   DATA[1768,11] := 19.63634;
   DATA[1768,12] := 2.208884;
   DATA[1768,13] := 823.5469;
   DATA[1768,14] := 1.0;
   DATA[1768,15] := 2.0;
   DATA[1768,16] := 1.0;
   DATA[1768,17] := 1.0;
   DATA[1768,18] := 1.0;
   DATA[1768,19] := 2.0;
   DATA[1768,20] := 148.808;
   DATA[1768,21] := 154.4219;
   DATA[1768,22] := 1.717105;
   DATA[1768,23] := 810.9075;
   DATA[1768,24] := 2.0;
   DATA[1768,25] := 2.0;
   DATA[1768,26] := 7.876058;
   DATA[1768,27] := 143.7067;
   DATA[1768,28] := 262.4007;
   DATA[1768,29] := 12.11228;
   DATA[1768,30] := 1.725455;
   DATA[1768,31] := 1.290124;
   DATA[1768,32] := 0.7353967;
   DATA[1768,33] := 0.3080421;
   DATA[1768,34] := 2.0;
   DATA[1768,35] := 250.1923;
   DATA[1768,36] := 1.681991;
   DATA[1768,37] := 188.974;
   DATA[1768,38] := 0.000128152;
   DATA[1768,39] := 1.0;
   DATA[1768,40] := 1.0;
   DATA[1769,0] := 2.554847;
   DATA[1769,1] := 822.777;
   DATA[1769,2] := 2.0;
   DATA[1769,3] := 1.0;
   DATA[1769,4] := 262.625;
   DATA[1769,5] := 8.46533;
   DATA[1769,6] := 319.7898;
   DATA[1769,8] := 1.0;
   DATA[1769,9] := 1.0;
   DATA[1769,10] := 1.0;
   DATA[1769,11] := 19.70037;
   DATA[1769,12] := 2.208884;
   DATA[1769,13] := 823.3466;
   DATA[1769,14] := 1.0;
   DATA[1769,15] := 2.0;
   DATA[1769,16] := 1.0;
   DATA[1769,17] := 1.0;
   DATA[1769,18] := 1.0;
   DATA[1769,19] := 2.0;
   DATA[1769,20] := 148.808;
   DATA[1769,21] := 154.4219;
   DATA[1769,22] := 1.717105;
   DATA[1769,23] := 810.6383;
   DATA[1769,24] := 2.0;
   DATA[1769,25] := 2.0;
   DATA[1769,26] := 7.876058;
   DATA[1769,27] := 143.7067;
   DATA[1769,28] := 262.4007;
   DATA[1769,29] := 12.11228;
   DATA[1769,30] := 1.725455;
   DATA[1769,31] := 1.291533;
   DATA[1769,32] := 0.7353967;
   DATA[1769,33] := 0.3083624;
   DATA[1769,34] := 2.0;
   DATA[1769,35] := 250.1923;
   DATA[1769,36] := 1.681991;
   DATA[1769,37] := 188.974;
   DATA[1769,38] := 0.000128152;
   DATA[1769,39] := 1.0;
   DATA[1769,40] := 1.0;
   DATA[1770,0] := 2.542036;
   DATA[1770,1] := 823.0518;
   DATA[1770,2] := 2.0;
   DATA[1770,3] := 1.0;
   DATA[1770,4] := 262.625;
   DATA[1770,5] := 8.46533;
   DATA[1770,6] := 319.7898;
   DATA[1770,8] := 1.0;
   DATA[1770,9] := 1.0;
   DATA[1770,10] := 1.0;
   DATA[1770,11] := 19.73558;
   DATA[1770,12] := 2.208884;
   DATA[1770,13] := 823.0262;
   DATA[1770,14] := 1.0;
   DATA[1770,15] := 2.0;
   DATA[1770,16] := 1.0;
   DATA[1770,17] := 1.0;
   DATA[1770,18] := 1.0;
   DATA[1770,19] := 2.0;
   DATA[1770,20] := 148.808;
   DATA[1770,21] := 154.3707;
   DATA[1770,22] := 1.717105;
   DATA[1770,23] := 811.0228;
   DATA[1770,24] := 2.0;
   DATA[1770,25] := 2.0;
   DATA[1770,26] := 7.876058;
   DATA[1770,27] := 143.5529;
   DATA[1770,28] := 262.4007;
   DATA[1770,29] := 12.11228;
   DATA[1770,30] := 1.725455;
   DATA[1770,31] := 1.291533;
   DATA[1770,32] := 0.7353967;
   DATA[1770,33] := 0.3084265;
   DATA[1770,34] := 2.0;
   DATA[1770,35] := 250.1923;
   DATA[1770,36] := 1.681991;
   DATA[1770,37] := 188.974;
   DATA[1770,38] := 0.000128152;
   DATA[1770,39] := 1.0;
   DATA[1770,40] := 1.0;
   DATA[1771,0] := 2.526022;
   DATA[1771,1] := 823.7976;
   DATA[1771,2] := 2.0;
   DATA[1771,3] := 1.0;
   DATA[1771,4] := 262.625;
   DATA[1771,5] := 8.46533;
   DATA[1771,6] := 319.7898;
   DATA[1771,8] := 1.0;
   DATA[1771,9] := 1.0;
   DATA[1771,10] := 1.0;
   DATA[1771,11] := 19.73558;
   DATA[1771,12] := 2.208884;
   DATA[1771,13] := 822.6657;
   DATA[1771,14] := 1.0;
   DATA[1771,15] := 2.0;
   DATA[1771,16] := 1.0;
   DATA[1771,17] := 1.0;
   DATA[1771,18] := 1.0;
   DATA[1771,19] := 2.0;
   DATA[1771,20] := 148.808;
   DATA[1771,21] := 154.3194;
   DATA[1771,22] := 1.716208;
   DATA[1771,23] := 810.9459;
   DATA[1771,24] := 2.0;
   DATA[1771,25] := 2.0;
   DATA[1771,26] := 7.876058;
   DATA[1771,27] := 143.5529;
   DATA[1771,28] := 262.4007;
   DATA[1771,29] := 12.11228;
   DATA[1771,30] := 1.725455;
   DATA[1771,31] := 1.291533;
   DATA[1771,32] := 0.7353967;
   DATA[1771,33] := 0.3084265;
   DATA[1771,34] := 2.0;
   DATA[1771,35] := 250.1923;
   DATA[1771,36] := 1.681991;
   DATA[1771,37] := 188.974;
   DATA[1771,38] := 0.000128152;
   DATA[1771,39] := 1.0;
   DATA[1771,40] := 1.0;
   DATA[1772,0] := 2.503923;
   DATA[1772,1] := 824.5042;
   DATA[1772,2] := 2.0;
   DATA[1772,3] := 1.0;
   DATA[1772,4] := 262.625;
   DATA[1772,5] := 8.46533;
   DATA[1772,6] := 319.7898;
   DATA[1772,8] := 1.0;
   DATA[1772,9] := 1.0;
   DATA[1772,10] := 1.0;
   DATA[1772,11] := 19.73558;
   DATA[1772,12] := 2.208884;
   DATA[1772,13] := 822.3853;
   DATA[1772,14] := 1.0;
   DATA[1772,15] := 2.0;
   DATA[1772,16] := 1.0;
   DATA[1772,17] := 1.0;
   DATA[1772,18] := 1.0;
   DATA[1772,19] := 2.0;
   DATA[1772,20] := 148.808;
   DATA[1772,21] := 154.2425;
   DATA[1772,22] := 1.715183;
   DATA[1772,23] := 811.4843;
   DATA[1772,24] := 2.0;
   DATA[1772,25] := 2.0;
   DATA[1772,26] := 7.876058;
   DATA[1772,27] := 143.5529;
   DATA[1772,28] := 262.4007;
   DATA[1772,29] := 12.11228;
   DATA[1772,30] := 1.723789;
   DATA[1772,31] := 1.282567;
   DATA[1772,32] := 0.7353967;
   DATA[1772,33] := 0.3084265;
   DATA[1772,34] := 2.0;
   DATA[1772,35] := 250.1923;
   DATA[1772,36] := 1.681991;
   DATA[1772,37] := 188.974;
   DATA[1772,38] := 0.000128152;
   DATA[1772,39] := 1.0;
   DATA[1772,40] := 1.0;
   DATA[1773,0] := 2.491432;
   DATA[1773,1] := 824.5042;
   DATA[1773,2] := 2.0;
   DATA[1773,3] := 1.0;
   DATA[1773,4] := 262.625;
   DATA[1773,5] := 8.46533;
   DATA[1773,6] := 319.7898;
   DATA[1773,8] := 1.0;
   DATA[1773,9] := 1.0;
   DATA[1773,10] := 1.0;
   DATA[1773,11] := 19.73558;
   DATA[1773,12] := 2.208884;
   DATA[1773,13] := 821.6643;
   DATA[1773,14] := 1.0;
   DATA[1773,15] := 2.0;
   DATA[1773,16] := 1.0;
   DATA[1773,17] := 1.0;
   DATA[1773,18] := 1.0;
   DATA[1773,19] := 2.0;
   DATA[1773,20] := 148.808;
   DATA[1773,21] := 154.2425;
   DATA[1773,22] := 1.715183;
   DATA[1773,23] := 811.3304;
   DATA[1773,24] := 2.0;
   DATA[1773,25] := 2.0;
   DATA[1773,26] := 7.876058;
   DATA[1773,27] := 143.5529;
   DATA[1773,28] := 262.4007;
   DATA[1773,29] := 12.11228;
   DATA[1773,30] := 1.723789;
   DATA[1773,31] := 1.266171;
   DATA[1773,32] := 0.7353967;
   DATA[1773,33] := 0.3084265;
   DATA[1773,34] := 2.0;
   DATA[1773,35] := 250.1923;
   DATA[1773,36] := 1.681991;
   DATA[1773,37] := 188.974;
   DATA[1773,38] := 0.000128152;
   DATA[1773,39] := 1.0;
   DATA[1773,40] := 1.0;
   DATA[1774,0] := 2.475098;
   DATA[1774,1] := 824.936;
   DATA[1774,2] := 2.0;
   DATA[1774,3] := 1.0;
   DATA[1774,4] := 262.625;
   DATA[1774,5] := 8.46533;
   DATA[1774,6] := 319.7898;
   DATA[1774,8] := 1.0;
   DATA[1774,9] := 1.0;
   DATA[1774,10] := 1.0;
   DATA[1774,11] := 19.73558;
   DATA[1774,12] := 2.208884;
   DATA[1774,13] := 821.8245;
   DATA[1774,14] := 1.0;
   DATA[1774,15] := 2.0;
   DATA[1774,16] := 1.0;
   DATA[1774,17] := 1.0;
   DATA[1774,18] := 1.0;
   DATA[1774,19] := 2.0;
   DATA[1774,20] := 148.808;
   DATA[1774,21] := 154.2425;
   DATA[1774,22] := 1.715183;
   DATA[1774,23] := 811.4073;
   DATA[1774,24] := 2.0;
   DATA[1774,25] := 2.0;
   DATA[1774,26] := 7.876058;
   DATA[1774,27] := 143.5529;
   DATA[1774,28] := 262.4007;
   DATA[1774,29] := 12.11228;
   DATA[1774,30] := 1.723789;
   DATA[1774,31] := 1.266299;
   DATA[1774,32] := 0.7353967;
   DATA[1774,33] := 0.3084265;
   DATA[1774,34] := 2.0;
   DATA[1774,35] := 250.032;
   DATA[1774,36] := 1.681991;
   DATA[1774,37] := 188.974;
   DATA[1774,38] := 0.000128152;
   DATA[1774,39] := 1.0;
   DATA[1774,40] := 1.0;
   DATA[1775,0] := 2.455241;
   DATA[1775,1] := 825.2892;
   DATA[1775,2] := 2.0;
   DATA[1775,3] := 1.0;
   DATA[1775,4] := 262.625;
   DATA[1775,5] := 8.46533;
   DATA[1775,6] := 319.7898;
   DATA[1775,8] := 1.0;
   DATA[1775,9] := 1.0;
   DATA[1775,10] := 1.0;
   DATA[1775,11] := 19.74198;
   DATA[1775,12] := 2.208884;
   DATA[1775,13] := 821.0235;
   DATA[1775,14] := 1.0;
   DATA[1775,15] := 2.0;
   DATA[1775,16] := 1.0;
   DATA[1775,17] := 1.0;
   DATA[1775,18] := 1.0;
   DATA[1775,19] := 2.0;
   DATA[1775,20] := 148.808;
   DATA[1775,21] := 154.5245;
   DATA[1775,22] := 1.715183;
   DATA[1775,23] := 811.4843;
   DATA[1775,24] := 2.0;
   DATA[1775,25] := 2.0;
   DATA[1775,26] := 7.876058;
   DATA[1775,27] := 143.5529;
   DATA[1775,28] := 262.4007;
   DATA[1775,29] := 12.11228;
   DATA[1775,30] := 1.723789;
   DATA[1775,31] := 1.260664;
   DATA[1775,32] := 0.7353967;
   DATA[1775,33] := 0.3084265;
   DATA[1775,34] := 2.0;
   DATA[1775,35] := 250.032;
   DATA[1775,36] := 1.762086;
   DATA[1775,37] := 188.9259;
   DATA[1775,38] := 0.000128152;
   DATA[1775,39] := 1.0;
   DATA[1775,40] := 1.0;
   DATA[1776,0] := 2.441149;
   DATA[1776,1] := 825.3677;
   DATA[1776,2] := 2.0;
   DATA[1776,3] := 1.0;
   DATA[1776,4] := 262.625;
   DATA[1776,5] := 8.46533;
   DATA[1776,6] := 319.7898;
   DATA[1776,8] := 1.0;
   DATA[1776,9] := 1.0;
   DATA[1776,10] := 1.0;
   DATA[1776,11] := 19.82201;
   DATA[1776,12] := 2.209013;
   DATA[1776,13] := 820.5428;
   DATA[1776,14] := 1.0;
   DATA[1776,15] := 2.0;
   DATA[1776,16] := 1.0;
   DATA[1776,17] := 1.0;
   DATA[1776,18] := 1.0;
   DATA[1776,19] := 2.0;
   DATA[1776,20] := 148.808;
   DATA[1776,21] := 154.5245;
   DATA[1776,22] := 1.718002;
   DATA[1776,23] := 811.1766;
   DATA[1776,24] := 2.0;
   DATA[1776,25] := 2.0;
   DATA[1776,26] := 7.876058;
   DATA[1776,27] := 143.5529;
   DATA[1776,28] := 262.5288;
   DATA[1776,29] := 12.11228;
   DATA[1776,30] := 1.723789;
   DATA[1776,31] := 1.265787;
   DATA[1776,32] := 0.7353967;
   DATA[1776,33] := 0.3084265;
   DATA[1776,34] := 2.0;
   DATA[1776,35] := 250.032;
   DATA[1776,36] := 1.810143;
   DATA[1776,37] := 188.9259;
   DATA[1776,38] := 0.000128152;
   DATA[1776,39] := 1.0;
   DATA[1776,40] := 1.0;
   DATA[1777,0] := 2.428658;
   DATA[1777,1] := 825.9173;
   DATA[1777,2] := 2.0;
   DATA[1777,3] := 1.0;
   DATA[1777,4] := 262.625;
   DATA[1777,5] := 8.46533;
   DATA[1777,6] := 319.7898;
   DATA[1777,8] := 1.0;
   DATA[1777,9] := 1.0;
   DATA[1777,10] := 1.0;
   DATA[1777,11] := 19.84762;
   DATA[1777,12] := 2.209013;
   DATA[1777,13] := 820.0622;
   DATA[1777,14] := 1.0;
   DATA[1777,15] := 2.0;
   DATA[1777,16] := 1.0;
   DATA[1777,17] := 1.0;
   DATA[1777,18] := 1.0;
   DATA[1777,19] := 2.0;
   DATA[1777,20] := 148.808;
   DATA[1777,21] := 154.5245;
   DATA[1777,22] := 1.718002;
   DATA[1777,23] := 811.5227;
   DATA[1777,24] := 2.0;
   DATA[1777,25] := 2.0;
   DATA[1777,26] := 7.876058;
   DATA[1777,27] := 143.5529;
   DATA[1777,28] := 262.5288;
   DATA[1777,29] := 12.11228;
   DATA[1777,30] := 1.723789;
   DATA[1777,31] := 1.267196;
   DATA[1777,32] := 0.7353967;
   DATA[1777,33] := 0.3084265;
   DATA[1777,34] := 2.0;
   DATA[1777,35] := 250.032;
   DATA[1777,36] := 1.810143;
   DATA[1777,37] := 188.9259;
   DATA[1777,38] := 0.000128152;
   DATA[1777,39] := 1.0;
   DATA[1777,40] := 1.0;
   DATA[1778,0] := 2.425135;
   DATA[1778,1] := 826.3491;
   DATA[1778,2] := 2.0;
   DATA[1778,3] := 1.0;
   DATA[1778,4] := 262.625;
   DATA[1778,5] := 8.46533;
   DATA[1778,6] := 319.7898;
   DATA[1778,8] := 1.0;
   DATA[1778,9] := 1.0;
   DATA[1778,10] := 1.0;
   DATA[1778,11] := 19.84762;
   DATA[1778,12] := 2.209525;
   DATA[1778,13] := 819.6216;
   DATA[1778,14] := 1.0;
   DATA[1778,15] := 2.0;
   DATA[1778,16] := 1.0;
   DATA[1778,17] := 1.0;
   DATA[1778,18] := 1.0;
   DATA[1778,19] := 2.0;
   DATA[1778,20] := 148.808;
   DATA[1778,21] := 154.5245;
   DATA[1778,22] := 1.718002;
   DATA[1778,23] := 811.0997;
   DATA[1778,24] := 2.0;
   DATA[1778,25] := 2.0;
   DATA[1778,26] := 7.876058;
   DATA[1778,27] := 143.5529;
   DATA[1778,28] := 262.5288;
   DATA[1778,29] := 12.11228;
   DATA[1778,30] := 1.723789;
   DATA[1778,31] := 1.262969;
   DATA[1778,32] := 0.7353967;
   DATA[1778,33] := 0.3084265;
   DATA[1778,34] := 2.0;
   DATA[1778,35] := 250.032;
   DATA[1778,36] := 1.810143;
   DATA[1778,37] := 188.9259;
   DATA[1778,38] := 0.000128152;
   DATA[1778,39] := 1.0;
   DATA[1778,40] := 1.0;
   DATA[1779,0] := 2.425135;
   DATA[1779,1] := 826.6631;
   DATA[1779,2] := 2.0;
   DATA[1779,3] := 1.0;
   DATA[1779,4] := 262.625;
   DATA[1779,5] := 8.46533;
   DATA[1779,6] := 319.7898;
   DATA[1779,8] := 1.0;
   DATA[1779,9] := 1.0;
   DATA[1779,10] := 1.0;
   DATA[1779,11] := 19.7836;
   DATA[1779,12] := 2.209525;
   DATA[1779,13] := 819.0208;
   DATA[1779,14] := 1.0;
   DATA[1779,15] := 2.0;
   DATA[1779,16] := 1.0;
   DATA[1779,17] := 1.0;
   DATA[1779,18] := 1.0;
   DATA[1779,19] := 2.0;
   DATA[1779,20] := 148.808;
   DATA[1779,21] := 154.5245;
   DATA[1779,22] := 1.718002;
   DATA[1779,23] := 810.7921;
   DATA[1779,24] := 2.0;
   DATA[1779,25] := 2.0;
   DATA[1779,26] := 7.876058;
   DATA[1779,27] := 143.5529;
   DATA[1779,28] := 262.5288;
   DATA[1779,29] := 12.11228;
   DATA[1779,30] := 1.723789;
   DATA[1779,31] := 1.267452;
   DATA[1779,32] := 0.7353967;
   DATA[1779,33] := 0.3084265;
   DATA[1779,34] := 2.0;
   DATA[1779,35] := 250.032;
   DATA[1779,36] := 1.665972;
   DATA[1779,37] := 188.9259;
   DATA[1779,38] := 0.000128152;
   DATA[1779,39] := 1.0;
   DATA[1779,40] := 1.0;
   DATA[1780,0] := 2.43026;
   DATA[1780,1] := 827.8799;
   DATA[1780,2] := 2.0;
   DATA[1780,3] := 1.0;
   DATA[1780,4] := 262.625;
   DATA[1780,5] := 8.46533;
   DATA[1780,6] := 319.7898;
   DATA[1780,8] := 1.0;
   DATA[1780,9] := 1.0;
   DATA[1780,10] := 1.0;
   DATA[1780,11] := 19.73558;
   DATA[1780,12] := 2.209525;
   DATA[1780,13] := 819.1409;
   DATA[1780,14] := 1.0;
   DATA[1780,15] := 2.0;
   DATA[1780,16] := 1.0;
   DATA[1780,17] := 1.0;
   DATA[1780,18] := 1.0;
   DATA[1780,19] := 2.0;
   DATA[1780,20] := 148.808;
   DATA[1780,21] := 154.5245;
   DATA[1780,22] := 1.715952;
   DATA[1780,23] := 811.0228;
   DATA[1780,24] := 2.0;
   DATA[1780,25] := 2.0;
   DATA[1780,26] := 7.876058;
   DATA[1780,27] := 143.5529;
   DATA[1780,28] := 262.5288;
   DATA[1780,29] := 12.11228;
   DATA[1780,30] := 1.723789;
   DATA[1780,31] := 1.28103;
   DATA[1780,32] := 0.7353967;
   DATA[1780,33] := 0.3084265;
   DATA[1780,34] := 2.0;
   DATA[1780,35] := 250.032;
   DATA[1780,36] := 1.665972;
   DATA[1780,37] := 188.8458;
   DATA[1780,38] := 0.000128152;
   DATA[1780,39] := 1.0;
   DATA[1780,40] := 1.0;
   DATA[1781,0] := 2.483105;
   DATA[1781,1] := 828.7042;
   DATA[1781,2] := 2.0;
   DATA[1781,3] := 1.0;
   DATA[1781,4] := 262.625;
   DATA[1781,5] := 8.46533;
   DATA[1781,6] := 319.7898;
   DATA[1781,8] := 1.0;
   DATA[1781,9] := 1.0;
   DATA[1781,10] := 1.0;
   DATA[1781,11] := 19.73558;
   DATA[1781,12] := 2.209525;
   DATA[1781,13] := 818.42;
   DATA[1781,14] := 1.0;
   DATA[1781,15] := 2.0;
   DATA[1781,16] := 1.0;
   DATA[1781,17] := 1.0;
   DATA[1781,18] := 1.0;
   DATA[1781,19] := 2.0;
   DATA[1781,20] := 148.808;
   DATA[1781,21] := 154.5245;
   DATA[1781,22] := 1.715952;
   DATA[1781,23] := 810.8306;
   DATA[1781,24] := 2.0;
   DATA[1781,25] := 2.0;
   DATA[1781,26] := 7.876058;
   DATA[1781,27] := 143.5529;
   DATA[1781,28] := 262.5288;
   DATA[1781,29] := 12.11228;
   DATA[1781,30] := 1.721738;
   DATA[1781,31] := 1.28167;
   DATA[1781,32] := 0.7353967;
   DATA[1781,33] := 0.3084265;
   DATA[1781,34] := 2.0;
   DATA[1781,35] := 250.032;
   DATA[1781,36] := 1.665972;
   DATA[1781,37] := 188.7337;
   DATA[1781,38] := 0.000128152;
   DATA[1781,39] := 1.0;
   DATA[1781,40] := 1.0;
   DATA[1782,0] := 2.519937;
   DATA[1782,1] := 829.2145;
   DATA[1782,2] := 2.0;
   DATA[1782,3] := 1.0;
   DATA[1782,4] := 262.625;
   DATA[1782,5] := 8.461164;
   DATA[1782,6] := 319.7898;
   DATA[1782,8] := 1.0;
   DATA[1782,9] := 1.0;
   DATA[1782,10] := 1.0;
   DATA[1782,11] := 19.73558;
   DATA[1782,12] := 2.209909;
   DATA[1782,13] := 818.0194;
   DATA[1782,14] := 1.0;
   DATA[1782,15] := 2.0;
   DATA[1782,16] := 1.0;
   DATA[1782,17] := 1.0;
   DATA[1782,18] := 1.0;
   DATA[1782,19] := 2.0;
   DATA[1782,20] := 148.808;
   DATA[1782,21] := 154.5245;
   DATA[1782,22] := 1.714029;
   DATA[1782,23] := 810.6383;
   DATA[1782,24] := 2.0;
   DATA[1782,25] := 2.0;
   DATA[1782,26] := 7.876058;
   DATA[1782,27] := 143.5529;
   DATA[1782,28] := 262.5288;
   DATA[1782,29] := 12.11228;
   DATA[1782,30] := 1.721738;
   DATA[1782,31] := 1.298322;
   DATA[1782,32] := 0.7353967;
   DATA[1782,33] := 0.3084265;
   DATA[1782,34] := 2.0;
   DATA[1782,35] := 249.7917;
   DATA[1782,36] := 1.665972;
   DATA[1782,37] := 188.7337;
   DATA[1782,38] := 0.000128152;
   DATA[1782,39] := 1.0;
   DATA[1782,40] := 1.0;
   DATA[1783,0] := 2.563174;
   DATA[1783,1] := 829.9211;
   DATA[1783,2] := 2.0;
   DATA[1783,3] := 1.0;
   DATA[1783,4] := 262.625;
   DATA[1783,5] := 8.460524;
   DATA[1783,6] := 319.7898;
   DATA[1783,8] := 1.0;
   DATA[1783,9] := 1.0;
   DATA[1783,10] := 1.0;
   DATA[1783,11] := 19.73558;
   DATA[1783,12] := 2.209909;
   DATA[1783,13] := 817.4186;
   DATA[1783,14] := 1.0;
   DATA[1783,15] := 2.0;
   DATA[1783,16] := 1.0;
   DATA[1783,17] := 1.0;
   DATA[1783,18] := 1.0;
   DATA[1783,19] := 2.0;
   DATA[1783,20] := 148.808;
   DATA[1783,21] := 154.5245;
   DATA[1783,22] := 1.712363;
   DATA[1783,23] := 810.7537;
   DATA[1783,24] := 2.0;
   DATA[1783,25] := 2.0;
   DATA[1783,26] := 7.876058;
   DATA[1783,27] := 143.5529;
   DATA[1783,28] := 262.5288;
   DATA[1783,29] := 12.11228;
   DATA[1783,30] := 1.721738;
   DATA[1783,31] := 1.295248;
   DATA[1783,32] := 0.7353967;
   DATA[1783,33] := 0.3084265;
   DATA[1783,34] := 2.0;
   DATA[1783,35] := 249.7597;
   DATA[1783,36] := 1.665972;
   DATA[1783,37] := 188.7337;
   DATA[1783,38] := 0.000128152;
   DATA[1783,39] := 1.0;
   DATA[1783,40] := 1.0;
   DATA[1784,0] := 2.596163;
   DATA[1784,1] := 830.3921;
   DATA[1784,2] := 2.0;
   DATA[1784,3] := 1.0;
   DATA[1784,4] := 262.625;
   DATA[1784,5] := 8.460524;
   DATA[1784,6] := 319.7898;
   DATA[1784,8] := 1.0;
   DATA[1784,9] := 1.0;
   DATA[1784,10] := 1.0;
   DATA[1784,11] := 19.65235;
   DATA[1784,12] := 2.209909;
   DATA[1784,13] := 817.4186;
   DATA[1784,14] := 1.0;
   DATA[1784,15] := 2.0;
   DATA[1784,16] := 1.0;
   DATA[1784,17] := 1.0;
   DATA[1784,18] := 1.0;
   DATA[1784,19] := 2.0;
   DATA[1784,20] := 148.808;
   DATA[1784,21] := 154.5245;
   DATA[1784,22] := 1.711723;
   DATA[1784,23] := 810.3691;
   DATA[1784,24] := 2.0;
   DATA[1784,25] := 2.0;
   DATA[1784,26] := 7.876058;
   DATA[1784,27] := 143.5529;
   DATA[1784,28] := 262.5288;
   DATA[1784,29] := 12.11228;
   DATA[1784,30] := 1.721738;
   DATA[1784,31] := 1.291149;
   DATA[1784,32] := 0.7353967;
   DATA[1784,33] := 0.3084265;
   DATA[1784,34] := 2.0;
   DATA[1784,35] := 249.7597;
   DATA[1784,36] := 1.665972;
   DATA[1784,37] := 188.7337;
   DATA[1784,38] := 0.000128152;
   DATA[1784,39] := 1.0;
   DATA[1784,40] := 1.0;
   DATA[1785,0] := 2.630112;
   DATA[1785,1] := 831.2949;
   DATA[1785,2] := 2.0;
   DATA[1785,3] := 1.0;
   DATA[1785,4] := 262.625;
   DATA[1785,5] := 8.460524;
   DATA[1785,6] := 319.7898;
   DATA[1785,8] := 1.0;
   DATA[1785,9] := 1.0;
   DATA[1785,10] := 1.0;
   DATA[1785,11] := 19.65235;
   DATA[1785,12] := 2.209909;
   DATA[1785,13] := 816.5775;
   DATA[1785,14] := 1.0;
   DATA[1785,15] := 2.0;
   DATA[1785,16] := 1.0;
   DATA[1785,17] := 1.0;
   DATA[1785,18] := 1.0;
   DATA[1785,19] := 2.0;
   DATA[1785,20] := 148.808;
   DATA[1785,21] := 154.5245;
   DATA[1785,22] := 1.711723;
   DATA[1785,23] := 810.5229;
   DATA[1785,24] := 2.0;
   DATA[1785,25] := 2.0;
   DATA[1785,26] := 7.876058;
   DATA[1785,27] := 143.5529;
   DATA[1785,28] := 262.5288;
   DATA[1785,29] := 11.92002;
   DATA[1785,30] := 1.721738;
   DATA[1785,31] := 1.298322;
   DATA[1785,32] := 0.7353967;
   DATA[1785,33] := 0.3084265;
   DATA[1785,34] := 2.0;
   DATA[1785,35] := 250.032;
   DATA[1785,36] := 1.665972;
   DATA[1785,37] := 188.7337;
   DATA[1785,38] := 0.000128152;
   DATA[1785,39] := 1.0;
   DATA[1785,40] := 1.0;
   DATA[1786,0] := 2.641963;
   DATA[1786,1] := 832.08;
   DATA[1786,2] := 2.0;
   DATA[1786,3] := 1.0;
   DATA[1786,4] := 262.625;
   DATA[1786,5] := 8.460524;
   DATA[1786,6] := 319.7898;
   DATA[1786,8] := 1.0;
   DATA[1786,9] := 1.0;
   DATA[1786,10] := 1.0;
   DATA[1786,11] := 19.61073;
   DATA[1786,12] := 2.209909;
   DATA[1786,13] := 816.3372;
   DATA[1786,14] := 1.0;
   DATA[1786,15] := 2.0;
   DATA[1786,16] := 1.0;
   DATA[1786,17] := 1.0;
   DATA[1786,18] := 1.0;
   DATA[1786,19] := 2.0;
   DATA[1786,20] := 148.808;
   DATA[1786,21] := 154.5245;
   DATA[1786,22] := 1.711723;
   DATA[1786,23] := 810.3691;
   DATA[1786,24] := 2.0;
   DATA[1786,25] := 2.0;
   DATA[1786,26] := 7.876058;
   DATA[1786,27] := 143.5529;
   DATA[1786,28] := 262.5288;
   DATA[1786,29] := 11.92002;
   DATA[1786,30] := 1.724173;
   DATA[1786,31] := 1.293326;
   DATA[1786,32] := 0.7353967;
   DATA[1786,33] := 0.3084265;
   DATA[1786,34] := 2.0;
   DATA[1786,35] := 250.032;
   DATA[1786,36] := 1.665972;
   DATA[1786,37] := 188.7337;
   DATA[1786,38] := 0.000128152;
   DATA[1786,39] := 1.0;
   DATA[1786,40] := 1.0;
   DATA[1787,0] := 2.649649;
   DATA[1787,1] := 832.551;
   DATA[1787,2] := 2.0;
   DATA[1787,3] := 1.0;
   DATA[1787,4] := 262.625;
   DATA[1787,5] := 8.460524;
   DATA[1787,6] := 319.7898;
   DATA[1787,8] := 1.0;
   DATA[1787,9] := 1.0;
   DATA[1787,10] := 1.0;
   DATA[1787,11] := 19.61073;
   DATA[1787,12] := 2.209909;
   DATA[1787,13] := 815.2557;
   DATA[1787,14] := 1.0;
   DATA[1787,15] := 2.0;
   DATA[1787,16] := 1.0;
   DATA[1787,17] := 1.0;
   DATA[1787,18] := 1.0;
   DATA[1787,19] := 2.0;
   DATA[1787,20] := 148.808;
   DATA[1787,21] := 154.5245;
   DATA[1787,22] := 1.711723;
   DATA[1787,23] := 810.7921;
   DATA[1787,24] := 2.0;
   DATA[1787,25] := 2.0;
   DATA[1787,26] := 7.876058;
   DATA[1787,27] := 143.5529;
   DATA[1787,28] := 262.5288;
   DATA[1787,29] := 11.92002;
   DATA[1787,30] := 1.724173;
   DATA[1787,31] := 1.281927;
   DATA[1787,32] := 0.7353967;
   DATA[1787,33] := 0.3084265;
   DATA[1787,34] := 2.0;
   DATA[1787,35] := 250.032;
   DATA[1787,36] := 1.665972;
   DATA[1787,37] := 188.8939;
   DATA[1787,38] := 0.000128152;
   DATA[1787,39] := 1.0;
   DATA[1787,40] := 1.0;
   DATA[1788,0] := 2.639721;
   DATA[1788,1] := 833.2576;
   DATA[1788,2] := 2.0;
   DATA[1788,3] := 1.0;
   DATA[1788,4] := 262.625;
   DATA[1788,5] := 8.460524;
   DATA[1788,6] := 319.7898;
   DATA[1788,8] := 1.0;
   DATA[1788,9] := 1.0;
   DATA[1788,10] := 1.0;
   DATA[1788,11] := 19.61073;
   DATA[1788,12] := 2.209909;
   DATA[1788,13] := 814.8151;
   DATA[1788,14] := 1.0;
   DATA[1788,15] := 2.0;
   DATA[1788,16] := 1.0;
   DATA[1788,17] := 1.0;
   DATA[1788,18] := 1.0;
   DATA[1788,19] := 2.0;
   DATA[1788,20] := 148.808;
   DATA[1788,21] := 154.5245;
   DATA[1788,22] := 1.711723;
   DATA[1788,23] := 810.7152;
   DATA[1788,24] := 2.0;
   DATA[1788,25] := 2.0;
   DATA[1788,26] := 7.876058;
   DATA[1788,27] := 143.5529;
   DATA[1788,28] := 262.3686;
   DATA[1788,29] := 11.92002;
   DATA[1788,30] := 1.724173;
   DATA[1788,31] := 1.28167;
   DATA[1788,32] := 0.7377012;
   DATA[1788,33] := 0.3084265;
   DATA[1788,34] := 2.0;
   DATA[1788,35] := 250.1442;
   DATA[1788,36] := 1.665972;
   DATA[1788,37] := 188.9259;
   DATA[1788,38] := 0.000128152;
   DATA[1788,39] := 1.0;
   DATA[1788,40] := 1.0;
   DATA[1789,0] := 2.618582;
   DATA[1789,1] := 833.7286;
   DATA[1789,2] := 2.0;
   DATA[1789,3] := 1.0;
   DATA[1789,4] := 262.625;
   DATA[1789,5] := 8.460524;
   DATA[1789,6] := 319.7898;
   DATA[1789,8] := 1.0;
   DATA[1789,9] := 1.0;
   DATA[1789,10] := 1.0;
   DATA[1789,11] := 19.65235;
   DATA[1789,12] := 2.209909;
   DATA[1789,13] := 813.974;
   DATA[1789,14] := 1.0;
   DATA[1789,15] := 2.0;
   DATA[1789,16] := 1.0;
   DATA[1789,17] := 1.0;
   DATA[1789,18] := 1.0;
   DATA[1789,19] := 2.0;
   DATA[1789,20] := 148.808;
   DATA[1789,21] := 154.5245;
   DATA[1789,22] := 1.714029;
   DATA[1789,23] := 810.4076;
   DATA[1789,24] := 2.0;
   DATA[1789,25] := 2.0;
   DATA[1789,26] := 7.876058;
   DATA[1789,27] := 143.5529;
   DATA[1789,28] := 262.3686;
   DATA[1789,29] := 11.92002;
   DATA[1789,30] := 1.724173;
   DATA[1789,31] := 1.281542;
   DATA[1789,32] := 0.7377012;
   DATA[1789,33] := 0.3084265;
   DATA[1789,34] := 2.0;
   DATA[1789,35] := 250.1762;
   DATA[1789,36] := 1.665972;
   DATA[1789,37] := 188.9419;
   DATA[1789,38] := 0.000128152;
   DATA[1789,39] := 1.0;
   DATA[1789,40] := 1.0;
   DATA[1790,0] := 2.609935;
   DATA[1790,1] := 834.4351;
   DATA[1790,2] := 2.0;
   DATA[1790,3] := 1.0;
   DATA[1790,4] := 262.625;
   DATA[1790,5] := 8.460524;
   DATA[1790,6] := 319.7898;
   DATA[1790,8] := 1.0;
   DATA[1790,9] := 1.0;
   DATA[1790,10] := 1.0;
   DATA[1790,11] := 19.67476;
   DATA[1790,12] := 2.209909;
   DATA[1790,13] := 814.014;
   DATA[1790,14] := 1.0;
   DATA[1790,15] := 2.0;
   DATA[1790,16] := 1.0;
   DATA[1790,17] := 1.0;
   DATA[1790,18] := 1.0;
   DATA[1790,19] := 2.0;
   DATA[1790,20] := 148.808;
   DATA[1790,21] := 154.5245;
   DATA[1790,22] := 1.714798;
   DATA[1790,23] := 810.9075;
   DATA[1790,24] := 2.0;
   DATA[1790,25] := 2.0;
   DATA[1790,26] := 7.876058;
   DATA[1790,27] := 143.5529;
   DATA[1790,28] := 262.3686;
   DATA[1790,29] := 11.92002;
   DATA[1790,30] := 1.726993;
   DATA[1790,31] := 1.288587;
   DATA[1790,32] := 0.7384694;
   DATA[1790,33] := 0.3084265;
   DATA[1790,34] := 2.0;
   DATA[1790,35] := 250.1762;
   DATA[1790,36] := 1.665972;
   DATA[1790,37] := 189.0541;
   DATA[1790,38] := 0.000128152;
   DATA[1790,39] := 1.0;
   DATA[1790,40] := 1.0;
   DATA[1791,0] := 2.603209;
   DATA[1791,1] := 834.9454;
   DATA[1791,2] := 2.0;
   DATA[1791,3] := 1.0;
   DATA[1791,4] := 262.625;
   DATA[1791,5] := 8.460524;
   DATA[1791,6] := 319.7898;
   DATA[1791,8] := 1.0;
   DATA[1791,9] := 1.0;
   DATA[1791,10] := 1.0;
   DATA[1791,11] := 19.68756;
   DATA[1791,12] := 2.209013;
   DATA[1791,13] := 813.5735;
   DATA[1791,14] := 1.0;
   DATA[1791,15] := 2.0;
   DATA[1791,16] := 1.0;
   DATA[1791,17] := 1.0;
   DATA[1791,18] := 1.0;
   DATA[1791,19] := 2.0;
   DATA[1791,20] := 148.808;
   DATA[1791,21] := 154.5245;
   DATA[1791,22] := 1.714798;
   DATA[1791,23] := 810.9075;
   DATA[1791,24] := 2.0;
   DATA[1791,25] := 2.0;
   DATA[1791,26] := 7.876058;
   DATA[1791,27] := 143.5529;
   DATA[1791,28] := 262.3686;
   DATA[1791,29] := 11.92002;
   DATA[1791,30] := 1.726993;
   DATA[1791,31] := 1.302037;
   DATA[1791,32] := 0.7387255;
   DATA[1791,33] := 0.3084265;
   DATA[1791,34] := 2.0;
   DATA[1791,35] := 250.1762;
   DATA[1791,36] := 1.665972;
   DATA[1791,37] := 189.0541;
   DATA[1791,38] := 0.000128152;
   DATA[1791,39] := 1.0;
   DATA[1791,40] := 1.0;
   DATA[1792,0] := 2.593281;
   DATA[1792,1] := 835.338;
   DATA[1792,2] := 2.0;
   DATA[1792,3] := 1.0;
   DATA[1792,4] := 262.625;
   DATA[1792,5] := 8.460524;
   DATA[1792,6] := 319.7898;
   DATA[1792,8] := 1.0;
   DATA[1792,9] := 1.0;
   DATA[1792,10] := 1.0;
   DATA[1792,11] := 19.73878;
   DATA[1792,12] := 2.209013;
   DATA[1792,13] := 813.5735;
   DATA[1792,14] := 1.0;
   DATA[1792,15] := 2.0;
   DATA[1792,16] := 1.0;
   DATA[1792,17] := 1.0;
   DATA[1792,18] := 1.0;
   DATA[1792,19] := 2.0;
   DATA[1792,20] := 148.808;
   DATA[1792,21] := 154.5245;
   DATA[1792,22] := 1.714798;
   DATA[1792,23] := 811.0997;
   DATA[1792,24] := 2.0;
   DATA[1792,25] := 2.0;
   DATA[1792,26] := 7.876058;
   DATA[1792,27] := 143.5529;
   DATA[1792,28] := 262.3686;
   DATA[1792,29] := 12.15073;
   DATA[1792,30] := 1.726993;
   DATA[1792,31] := 1.302037;
   DATA[1792,32] := 0.7387255;
   DATA[1792,33] := 0.3084265;
   DATA[1792,34] := 2.0;
   DATA[1792,35] := 250.1762;
   DATA[1792,36] := 1.665972;
   DATA[1792,37] := 189.0541;
   DATA[1792,38] := 0.000128152;
   DATA[1792,39] := 1.0;
   DATA[1792,40] := 1.0;
   DATA[1793,0] := 2.56926;
   DATA[1793,1] := 836.0052;
   DATA[1793,2] := 2.0;
   DATA[1793,3] := 1.0;
   DATA[1793,4] := 262.625;
   DATA[1793,5] := 8.460524;
   DATA[1793,6] := 319.7898;
   DATA[1793,8] := 1.0;
   DATA[1793,9] := 1.0;
   DATA[1793,10] := 1.0;
   DATA[1793,11] := 19.73878;
   DATA[1793,12] := 2.209013;
   DATA[1793,13] := 812.9326;
   DATA[1793,14] := 1.0;
   DATA[1793,15] := 2.0;
   DATA[1793,16] := 1.0;
   DATA[1793,17] := 1.0;
   DATA[1793,18] := 1.0;
   DATA[1793,19] := 2.0;
   DATA[1793,20] := 148.808;
   DATA[1793,21] := 154.7039;
   DATA[1793,22] := 1.714798;
   DATA[1793,23] := 811.292;
   DATA[1793,24] := 2.0;
   DATA[1793,25] := 2.0;
   DATA[1793,26] := 7.876058;
   DATA[1793,27] := 143.5529;
   DATA[1793,28] := 262.3686;
   DATA[1793,29] := 12.15073;
   DATA[1793,30] := 1.726993;
   DATA[1793,31] := 1.302037;
   DATA[1793,32] := 0.7361649;
   DATA[1793,33] := 0.3084265;
   DATA[1793,34] := 2.0;
   DATA[1793,35] := 250.1762;
   DATA[1793,36] := 1.665972;
   DATA[1793,37] := 189.0541;
   DATA[1793,38] := 0.000128152;
   DATA[1793,39] := 1.0;
   DATA[1793,40] := 1.0;
   DATA[1794,0] := 2.554527;
   DATA[1794,1] := 836.1622;
   DATA[1794,2] := 2.0;
   DATA[1794,3] := 1.0;
   DATA[1794,4] := 262.625;
   DATA[1794,5] := 8.460524;
   DATA[1794,6] := 319.8154;
   DATA[1794,8] := 1.0;
   DATA[1794,9] := 1.0;
   DATA[1794,10] := 1.0;
   DATA[1794,11] := 19.73878;
   DATA[1794,12] := 2.209013;
   DATA[1794,13] := 812.452;
   DATA[1794,14] := 1.0;
   DATA[1794,15] := 2.0;
   DATA[1794,16] := 1.0;
   DATA[1794,17] := 1.0;
   DATA[1794,18] := 1.0;
   DATA[1794,19] := 2.0;
   DATA[1794,20] := 148.808;
   DATA[1794,21] := 154.7039;
   DATA[1794,22] := 1.71467;
   DATA[1794,23] := 810.8306;
   DATA[1794,24] := 2.0;
   DATA[1794,25] := 2.0;
   DATA[1794,26] := 7.876058;
   DATA[1794,27] := 143.5529;
   DATA[1794,28] := 262.3686;
   DATA[1794,29] := 12.15073;
   DATA[1794,30] := 1.726993;
   DATA[1794,31] := 1.302037;
   DATA[1794,32] := 0.7357808;
   DATA[1794,33] := 0.3084265;
   DATA[1794,34] := 2.0;
   DATA[1794,35] := 250.1762;
   DATA[1794,36] := 1.665972;
   DATA[1794,37] := 189.0541;
   DATA[1794,38] := 0.000128152;
   DATA[1794,39] := 1.0;
   DATA[1794,40] := 1.0;
   DATA[1795,0] := 2.538833;
   DATA[1795,1] := 836.3585;
   DATA[1795,2] := 2.0;
   DATA[1795,3] := 1.0;
   DATA[1795,4] := 262.625;
   DATA[1795,5] := 8.460524;
   DATA[1795,6] := 319.8667;
   DATA[1795,8] := 1.0;
   DATA[1795,9] := 1.0;
   DATA[1795,10] := 1.0;
   DATA[1795,11] := 19.73878;
   DATA[1795,12] := 2.209013;
   DATA[1795,13] := 812.0114;
   DATA[1795,14] := 1.0;
   DATA[1795,15] := 2.0;
   DATA[1795,16] := 1.0;
   DATA[1795,17] := 1.0;
   DATA[1795,18] := 1.0;
   DATA[1795,19] := 2.0;
   DATA[1795,20] := 148.808;
   DATA[1795,21] := 154.7039;
   DATA[1795,22] := 1.713261;
   DATA[1795,23] := 811.0997;
   DATA[1795,24] := 2.0;
   DATA[1795,25] := 2.0;
   DATA[1795,26] := 7.876058;
   DATA[1795,27] := 143.5529;
   DATA[1795,28] := 262.3686;
   DATA[1795,29] := 12.15073;
   DATA[1795,30] := 1.726993;
   DATA[1795,31] := 1.302037;
   DATA[1795,32] := 0.7351407;
   DATA[1795,33] := 0.3084265;
   DATA[1795,34] := 2.0;
   DATA[1795,35] := 250.1762;
   DATA[1795,36] := 1.665972;
   DATA[1795,37] := 189.0541;
   DATA[1795,38] := 0.000128152;
   DATA[1795,39] := 1.0;
   DATA[1795,40] := 1.0;
   DATA[1796,0] := 2.524101;
   DATA[1796,1] := 836.3978;
   DATA[1796,2] := 2.0;
   DATA[1796,3] := 1.0;
   DATA[1796,4] := 262.625;
   DATA[1796,5] := 8.462767;
   DATA[1796,6] := 319.8667;
   DATA[1796,8] := 1.0;
   DATA[1796,9] := 1.0;
   DATA[1796,10] := 1.0;
   DATA[1796,11] := 19.73878;
   DATA[1796,12] := 2.207731;
   DATA[1796,13] := 811.1302;
   DATA[1796,14] := 1.0;
   DATA[1796,15] := 2.0;
   DATA[1796,16] := 1.0;
   DATA[1796,17] := 1.0;
   DATA[1796,18] := 1.0;
   DATA[1796,19] := 2.0;
   DATA[1796,20] := 148.808;
   DATA[1796,21] := 154.5501;
   DATA[1796,22] := 1.713261;
   DATA[1796,23] := 810.7537;
   DATA[1796,24] := 2.0;
   DATA[1796,25] := 2.0;
   DATA[1796,26] := 7.876058;
   DATA[1796,27] := 143.5529;
   DATA[1796,28] := 262.3686;
   DATA[1796,29] := 12.15073;
   DATA[1796,30] := 1.726993;
   DATA[1796,31] := 1.302037;
   DATA[1796,32] := 0.7351407;
   DATA[1796,33] := 0.3084265;
   DATA[1796,34] := 2.0;
   DATA[1796,35] := 250.1762;
   DATA[1796,36] := 1.665972;
   DATA[1796,37] := 188.974;
   DATA[1796,38] := 0.000128152;
   DATA[1796,39] := 1.0;
   DATA[1796,40] := 1.0;
   DATA[1797,0] := 2.506485;
   DATA[1797,1] := 836.3978;
   DATA[1797,2] := 2.0;
   DATA[1797,3] := 1.0;
   DATA[1797,4] := 262.625;
   DATA[1797,5] := 8.462767;
   DATA[1797,6] := 319.8667;
   DATA[1797,8] := 1.0;
   DATA[1797,9] := 1.0;
   DATA[1797,10] := 1.0;
   DATA[1797,11] := 19.73878;
   DATA[1797,12] := 2.207731;
   DATA[1797,13] := 810.8498;
   DATA[1797,14] := 1.0;
   DATA[1797,15] := 2.0;
   DATA[1797,16] := 1.0;
   DATA[1797,17] := 1.0;
   DATA[1797,18] := 1.0;
   DATA[1797,19] := 2.0;
   DATA[1797,20] := 148.808;
   DATA[1797,21] := 154.5501;
   DATA[1797,22] := 1.713261;
   DATA[1797,23] := 810.7921;
   DATA[1797,24] := 2.0;
   DATA[1797,25] := 2.0;
   DATA[1797,26] := 7.876058;
   DATA[1797,27] := 143.3479;
   DATA[1797,28] := 262.3686;
   DATA[1797,29] := 12.15073;
   DATA[1797,30] := 1.726993;
   DATA[1797,31] := 1.293455;
   DATA[1797,32] := 0.7351407;
   DATA[1797,33] := 0.3084265;
   DATA[1797,34] := 2.0;
   DATA[1797,35] := 250.1762;
   DATA[1797,36] := 1.665972;
   DATA[1797,37] := 188.974;
   DATA[1797,38] := 0.000128152;
   DATA[1797,39] := 1.0;
   DATA[1797,40] := 1.0;
   DATA[1798,0] := 2.493675;
   DATA[1798,1] := 836.7118;
   DATA[1798,2] := 2.0;
   DATA[1798,3] := 1.0;
   DATA[1798,4] := 262.625;
   DATA[1798,5] := 8.462767;
   DATA[1798,6] := 319.8667;
   DATA[1798,8] := 1.0;
   DATA[1798,9] := 1.0;
   DATA[1798,10] := 1.0;
   DATA[1798,11] := 19.67155;
   DATA[1798,12] := 2.207731;
   DATA[1798,13] := 810.4092;
   DATA[1798,14] := 1.0;
   DATA[1798,15] := 2.0;
   DATA[1798,16] := 1.0;
   DATA[1798,17] := 1.0;
   DATA[1798,18] := 1.0;
   DATA[1798,19] := 2.0;
   DATA[1798,20] := 148.808;
   DATA[1798,21] := 154.5501;
   DATA[1798,22] := 1.71467;
   DATA[1798,23] := 810.5999;
   DATA[1798,24] := 2.0;
   DATA[1798,25] := 2.0;
   DATA[1798,26] := 7.876058;
   DATA[1798,27] := 143.3479;
   DATA[1798,28] := 262.3686;
   DATA[1798,29] := 12.15073;
   DATA[1798,30] := 1.726993;
   DATA[1798,31] := 1.292046;
   DATA[1798,32] := 0.7351407;
   DATA[1798,33] := 0.3084265;
   DATA[1798,34] := 2.0;
   DATA[1798,35] := 250.1762;
   DATA[1798,36] := 1.665972;
   DATA[1798,37] := 188.974;
   DATA[1798,38] := 0.000128152;
   DATA[1798,39] := 1.0;
   DATA[1798,40] := 1.0;
   DATA[1799,0] := 2.477981;
   DATA[1799,1] := 837.2614;
   DATA[1799,2] := 2.0;
   DATA[1799,3] := 1.0;
   DATA[1799,4] := 262.625;
   DATA[1799,5] := 8.462767;
   DATA[1799,6] := 319.8667;
   DATA[1799,8] := 1.0;
   DATA[1799,9] := 1.0;
   DATA[1799,10] := 1.0;
   DATA[1799,11] := 19.67155;
   DATA[1799,12] := 2.207731;
   DATA[1799,13] := 810.2089;
   DATA[1799,14] := 1.0;
   DATA[1799,15] := 2.0;
   DATA[1799,16] := 1.0;
   DATA[1799,17] := 1.0;
   DATA[1799,18] := 1.0;
   DATA[1799,19] := 2.0;
   DATA[1799,20] := 148.808;
   DATA[1799,21] := 154.5501;
   DATA[1799,22] := 1.716592;
   DATA[1799,23] := 810.9844;
   DATA[1799,24] := 2.0;
   DATA[1799,25] := 2.0;
   DATA[1799,26] := 7.874135;
   DATA[1799,27] := 143.3479;
   DATA[1799,28] := 262.3686;
   DATA[1799,29] := 12.15073;
   DATA[1799,30] := 1.726737;
   DATA[1799,31] := 1.290893;
   DATA[1799,32] := 0.7351407;
   DATA[1799,33] := 0.3084265;
   DATA[1799,34] := 2.0;
   DATA[1799,35] := 250.1762;
   DATA[1799,36] := 1.665972;
   DATA[1799,37] := 188.974;
   DATA[1799,38] := 0.000128152;
   DATA[1799,39] := 1.0;
   DATA[1799,40] := 1.0;
   DATA[1800,0] := 2.462287;
   DATA[1800,1] := 837.6539;
   DATA[1800,2] := 2.0;
   DATA[1800,3] := 1.0;
   DATA[1800,4] := 262.625;
   DATA[1800,5] := 8.462767;
   DATA[1800,6] := 319.8667;
   DATA[1800,8] := 1.0;
   DATA[1800,9] := 1.0;
   DATA[1800,10] := 1.0;
   DATA[1800,11] := 19.67155;
   DATA[1800,12] := 2.208372;
   DATA[1800,13] := 810.4493;
   DATA[1800,14] := 1.0;
   DATA[1800,15] := 2.0;
   DATA[1800,16] := 1.0;
   DATA[1800,17] := 1.0;
   DATA[1800,18] := 1.0;
   DATA[1800,19] := 2.0;
   DATA[1800,20] := 148.808;
   DATA[1800,21] := 154.5501;
   DATA[1800,22] := 1.717105;
   DATA[1800,23] := 810.7921;
   DATA[1800,24] := 2.0;
   DATA[1800,25] := 2.0;
   DATA[1800,26] := 7.872853;
   DATA[1800,27] := 143.3479;
   DATA[1800,28] := 262.3686;
   DATA[1800,29] := 12.15073;
   DATA[1800,30] := 1.726737;
   DATA[1800,31] := 1.282311;
   DATA[1800,32] := 0.7351407;
   DATA[1800,33] := 0.3084265;
   DATA[1800,34] := 2.0;
   DATA[1800,35] := 250.1762;
   DATA[1800,36] := 1.665972;
   DATA[1800,37] := 188.974;
   DATA[1800,38] := 0.000128152;
   DATA[1800,39] := 1.0;
   DATA[1800,40] := 1.0;
   DATA[1801,0] := 2.447234;
   DATA[1801,1] := 838.2427;
   DATA[1801,2] := 2.0;
   DATA[1801,3] := 1.0;
   DATA[1801,4] := 262.625;
   DATA[1801,5] := 8.462767;
   DATA[1801,6] := 319.8667;
   DATA[1801,8] := 1.0;
   DATA[1801,9] := 1.0;
   DATA[1801,10] := 1.0;
   DATA[1801,11] := 19.67155;
   DATA[1801,12] := 2.208884;
   DATA[1801,13] := 809.8484;
   DATA[1801,14] := 1.0;
   DATA[1801,15] := 2.0;
   DATA[1801,16] := 1.0;
   DATA[1801,17] := 1.0;
   DATA[1801,18] := 1.0;
   DATA[1801,19] := 2.0;
   DATA[1801,20] := 148.808;
   DATA[1801,21] := 154.5501;
   DATA[1801,22] := 1.717105;
   DATA[1801,23] := 810.3691;
   DATA[1801,24] := 2.0;
   DATA[1801,25] := 2.0;
   DATA[1801,26] := 7.872853;
   DATA[1801,27] := 143.3479;
   DATA[1801,28] := 262.3686;
   DATA[1801,29] := 12.15073;
   DATA[1801,30] := 1.726737;
   DATA[1801,31] := 1.288843;
   DATA[1801,32] := 0.7351407;
   DATA[1801,33] := 0.3084265;
   DATA[1801,34] := 2.0;
   DATA[1801,35] := 250.1762;
   DATA[1801,36] := 1.665972;
   DATA[1801,37] := 189.1022;
   DATA[1801,38] := 0.000128152;
   DATA[1801,39] := 1.0;
   DATA[1801,40] := 1.0;
   DATA[1802,0] := 2.432181;
   DATA[1802,1] := 838.6744;
   DATA[1802,2] := 2.0;
   DATA[1802,3] := 1.0;
   DATA[1802,4] := 262.625;
   DATA[1802,5] := 8.463728;
   DATA[1802,6] := 319.8667;
   DATA[1802,8] := 1.0;
   DATA[1802,9] := 1.0;
   DATA[1802,10] := 1.0;
   DATA[1802,11] := 19.67155;
   DATA[1802,12] := 2.208884;
   DATA[1802,13] := 809.6082;
   DATA[1802,14] := 1.0;
   DATA[1802,15] := 2.0;
   DATA[1802,16] := 1.0;
   DATA[1802,17] := 1.0;
   DATA[1802,18] := 1.0;
   DATA[1802,19] := 2.0;
   DATA[1802,20] := 148.808;
   DATA[1802,21] := 154.5501;
   DATA[1802,22] := 1.717105;
   DATA[1802,23] := 810.3307;
   DATA[1802,24] := 2.0;
   DATA[1802,25] := 2.0;
   DATA[1802,26] := 7.872853;
   DATA[1802,27] := 143.3479;
   DATA[1802,28] := 262.3686;
   DATA[1802,29] := 12.15073;
   DATA[1802,30] := 1.725583;
   DATA[1802,31] := 1.292046;
   DATA[1802,32] := 0.7351407;
   DATA[1802,33] := 0.3084265;
   DATA[1802,34] := 2.0;
   DATA[1802,35] := 250.1762;
   DATA[1802,36] := 1.665972;
   DATA[1802,37] := 189.1022;
   DATA[1802,38] := 0.000128152;
   DATA[1802,39] := 1.0;
   DATA[1802,40] := 1.0;
   DATA[1803,0] := 2.428018;
   DATA[1803,1] := 839.3025;
   DATA[1803,2] := 2.0;
   DATA[1803,3] := 1.0;
   DATA[1803,4] := 262.625;
   DATA[1803,5] := 8.46533;
   DATA[1803,6] := 320.0461;
   DATA[1803,8] := 1.0;
   DATA[1803,9] := 1.0;
   DATA[1803,10] := 1.0;
   DATA[1803,11] := 19.67155;
   DATA[1803,12] := 2.208884;
   DATA[1803,13] := 809.2476;
   DATA[1803,14] := 1.0;
   DATA[1803,15] := 2.0;
   DATA[1803,16] := 1.0;
   DATA[1803,17] := 1.0;
   DATA[1803,18] := 1.0;
   DATA[1803,19] := 2.0;
   DATA[1803,20] := 148.808;
   DATA[1803,21] := 154.5501;
   DATA[1803,22] := 1.717105;
   DATA[1803,23] := 810.2922;
   DATA[1803,24] := 2.0;
   DATA[1803,25] := 2.0;
   DATA[1803,26] := 7.872853;
   DATA[1803,27] := 143.3222;
   DATA[1803,28] := 262.3686;
   DATA[1803,29] := 12.15073;
   DATA[1803,30] := 1.724814;
   DATA[1803,31] := 1.286282;
   DATA[1803,32] := 0.7351407;
   DATA[1803,33] := 0.3084265;
   DATA[1803,34] := 2.0;
   DATA[1803,35] := 250.1762;
   DATA[1803,36] := 1.665972;
   DATA[1803,37] := 189.1022;
   DATA[1803,38] := 0.000128152;
   DATA[1803,39] := 1.0;
   DATA[1803,40] := 1.0;
   DATA[1804,0] := 2.428018;
   DATA[1804,1] := 839.3025;
   DATA[1804,2] := 2.0;
   DATA[1804,3] := 1.0;
   DATA[1804,4] := 262.625;
   DATA[1804,5] := 8.46533;
   DATA[1804,6] := 320.0461;
   DATA[1804,8] := 1.0;
   DATA[1804,9] := 1.0;
   DATA[1804,10] := 1.0;
   DATA[1804,11] := 19.73238;
   DATA[1804,12] := 2.208884;
   DATA[1804,13] := 808.5267;
   DATA[1804,14] := 1.0;
   DATA[1804,15] := 2.0;
   DATA[1804,16] := 1.0;
   DATA[1804,17] := 1.0;
   DATA[1804,18] := 1.0;
   DATA[1804,19] := 2.0;
   DATA[1804,20] := 148.808;
   DATA[1804,21] := 154.5501;
   DATA[1804,22] := 1.717105;
   DATA[1804,23] := 810.5614;
   DATA[1804,24] := 2.0;
   DATA[1804,25] := 2.0;
   DATA[1804,26] := 7.872853;
   DATA[1804,27] := 143.3222;
   DATA[1804,28] := 262.3686;
   DATA[1804,29] := 12.15073;
   DATA[1804,30] := 1.724814;
   DATA[1804,31] := 1.286282;
   DATA[1804,32] := 0.7351407;
   DATA[1804,33] := 0.3084265;
   DATA[1804,34] := 2.0;
   DATA[1804,35] := 250.1762;
   DATA[1804,36] := 1.665972;
   DATA[1804,37] := 189.0861;
   DATA[1804,38] := 0.000128152;
   DATA[1804,39] := 1.0;
   DATA[1804,40] := 1.0;
   DATA[1805,0] := 2.444031;
   DATA[1805,1] := 839.695;
   DATA[1805,2] := 2.0;
   DATA[1805,3] := 1.0;
   DATA[1805,4] := 262.625;
   DATA[1805,5] := 8.46533;
   DATA[1805,6] := 320.0461;
   DATA[1805,8] := 1.0;
   DATA[1805,9] := 1.0;
   DATA[1805,10] := 1.0;
   DATA[1805,11] := 19.73558;
   DATA[1805,12] := 2.208884;
   DATA[1805,13] := 808.5267;
   DATA[1805,14] := 1.0;
   DATA[1805,15] := 2.0;
   DATA[1805,16] := 1.0;
   DATA[1805,17] := 1.0;
   DATA[1805,18] := 1.0;
   DATA[1805,19] := 2.0;
   DATA[1805,20] := 148.808;
   DATA[1805,21] := 154.5501;
   DATA[1805,22] := 1.717105;
   DATA[1805,23] := 810.6383;
   DATA[1805,24] := 2.0;
   DATA[1805,25] := 2.0;
   DATA[1805,26] := 7.872853;
   DATA[1805,27] := 143.3222;
   DATA[1805,28] := 262.3686;
   DATA[1805,29] := 12.15073;
   DATA[1805,30] := 1.724814;
   DATA[1805,31] := 1.283592;
   DATA[1805,32] := 0.7351407;
   DATA[1805,33] := 0.3084265;
   DATA[1805,34] := 2.0;
   DATA[1805,35] := 250.1762;
   DATA[1805,36] := 1.665972;
   DATA[1805,37] := 189.006;
   DATA[1805,38] := 0.000128152;
   DATA[1805,39] := 1.0;
   DATA[1805,40] := 1.0;
   DATA[1806,0] := 2.496237;
   DATA[1806,1] := 839.3025;
   DATA[1806,2] := 2.0;
   DATA[1806,3] := 1.0;
   DATA[1806,4] := 262.625;
   DATA[1806,5] := 8.46533;
   DATA[1806,6] := 320.0461;
   DATA[1806,8] := 1.0;
   DATA[1806,9] := 1.0;
   DATA[1806,10] := 1.0;
   DATA[1806,11] := 19.75159;
   DATA[1806,12] := 2.208884;
   DATA[1806,13] := 808.3665;
   DATA[1806,14] := 1.0;
   DATA[1806,15] := 2.0;
   DATA[1806,16] := 1.0;
   DATA[1806,17] := 1.0;
   DATA[1806,18] := 1.0;
   DATA[1806,19] := 2.0;
   DATA[1806,20] := 148.808;
   DATA[1806,21] := 154.5501;
   DATA[1806,22] := 1.715824;
   DATA[1806,23] := 810.5999;
   DATA[1806,24] := 2.0;
   DATA[1806,25] := 2.0;
   DATA[1806,26] := 7.872853;
   DATA[1806,27] := 143.3222;
   DATA[1806,28] := 262.3686;
   DATA[1806,29] := 12.15073;
   DATA[1806,30] := 1.724814;
   DATA[1806,31] := 1.271423;
   DATA[1806,32] := 0.7351407;
   DATA[1806,33] := 0.3084265;
   DATA[1806,34] := 2.0;
   DATA[1806,35] := 250.1762;
   DATA[1806,36] := 1.665972;
   DATA[1806,37] := 189.006;
   DATA[1806,38] := 0.000128152;
   DATA[1806,39] := 1.0;
   DATA[1806,40] := 1.0;
   DATA[1807,0] := 2.528264;
   DATA[1807,1] := 840.0483;
   DATA[1807,2] := 2.0;
   DATA[1807,3] := 1.0;
   DATA[1807,4] := 262.625;
   DATA[1807,5] := 8.46533;
   DATA[1807,6] := 320.0461;
   DATA[1807,8] := 1.0;
   DATA[1807,9] := 1.0;
   DATA[1807,10] := 1.0;
   DATA[1807,11] := 19.70677;
   DATA[1807,12] := 2.208628;
   DATA[1807,13] := 807.1248;
   DATA[1807,14] := 1.0;
   DATA[1807,15] := 2.0;
   DATA[1807,16] := 1.0;
   DATA[1807,17] := 1.0;
   DATA[1807,18] := 1.0;
   DATA[1807,19] := 2.0;
   DATA[1807,20] := 148.808;
   DATA[1807,21] := 154.5501;
   DATA[1807,22] := 1.715567;
   DATA[1807,23] := 810.9844;
   DATA[1807,24] := 2.0;
   DATA[1807,25] := 2.0;
   DATA[1807,26] := 7.874455;
   DATA[1807,27] := 143.3222;
   DATA[1807,28] := 262.3686;
   DATA[1807,29] := 12.15073;
   DATA[1807,30] := 1.724814;
   DATA[1807,31] := 1.271295;
   DATA[1807,32] := 0.7351407;
   DATA[1807,33] := 0.3084265;
   DATA[1807,34] := 2.0;
   DATA[1807,35] := 250.2563;
   DATA[1807,36] := 1.69801;
   DATA[1807,37] := 189.006;
   DATA[1807,38] := 0.000128152;
   DATA[1807,39] := 1.0;
   DATA[1807,40] := 1.0;
   DATA[1808,0] := 2.575345;
   DATA[1808,1] := 840.7941;
   DATA[1808,2] := 2.0;
   DATA[1808,3] := 1.0;
   DATA[1808,4] := 262.625;
   DATA[1808,5] := 8.46533;
   DATA[1808,6] := 320.0461;
   DATA[1808,8] := 1.0;
   DATA[1808,9] := 1.0;
   DATA[1808,10] := 1.0;
   DATA[1808,11] := 19.66835;
   DATA[1808,12] := 2.207731;
   DATA[1808,13] := 806.564;
   DATA[1808,14] := 1.0;
   DATA[1808,15] := 2.0;
   DATA[1808,16] := 1.0;
   DATA[1808,17] := 1.0;
   DATA[1808,18] := 1.0;
   DATA[1808,19] := 2.0;
   DATA[1808,20] := 148.808;
   DATA[1808,21] := 154.5501;
   DATA[1808,22] := 1.715567;
   DATA[1808,23] := 810.7921;
   DATA[1808,24] := 2.0;
   DATA[1808,25] := 2.0;
   DATA[1808,26] := 7.874455;
   DATA[1808,27] := 143.3222;
   DATA[1808,28] := 262.3686;
   DATA[1808,29] := 12.15073;
   DATA[1808,30] := 1.726737;
   DATA[1808,31] := 1.271295;
   DATA[1808,32] := 0.7351407;
   DATA[1808,33] := 0.3075937;
   DATA[1808,34] := 2.0;
   DATA[1808,35] := 250.4005;
   DATA[1808,36] := 1.69801;
   DATA[1808,37] := 189.2143;
   DATA[1808,38] := 0.000128152;
   DATA[1808,39] := 1.0;
   DATA[1808,40] := 1.0;
   DATA[1809,0] := 2.60481;
   DATA[1809,1] := 841.4221;
   DATA[1809,2] := 2.0;
   DATA[1809,3] := 1.0;
   DATA[1809,4] := 262.625;
   DATA[1809,5] := 8.46533;
   DATA[1809,6] := 320.0461;
   DATA[1809,8] := 1.0;
   DATA[1809,9] := 1.0;
   DATA[1809,10] := 1.0;
   DATA[1809,11] := 19.66835;
   DATA[1809,12] := 2.207091;
   DATA[1809,13] := 805.6027;
   DATA[1809,14] := 1.0;
   DATA[1809,15] := 2.0;
   DATA[1809,16] := 1.0;
   DATA[1809,17] := 1.0;
   DATA[1809,18] := 1.0;
   DATA[1809,19] := 2.0;
   DATA[1809,20] := 148.808;
   DATA[1809,21] := 154.5501;
   DATA[1809,22] := 1.717105;
   DATA[1809,23] := 811.0997;
   DATA[1809,24] := 2.0;
   DATA[1809,25] := 2.0;
   DATA[1809,26] := 7.874455;
   DATA[1809,27] := 143.3222;
   DATA[1809,28] := 262.3686;
   DATA[1809,29] := 12.15073;
   DATA[1809,30] := 1.726737;
   DATA[1809,31] := 1.28372;
   DATA[1809,32] := 0.7351407;
   DATA[1809,33] := 0.306761;
   DATA[1809,34] := 2.0;
   DATA[1809,35] := 250.4005;
   DATA[1809,36] := 1.69801;
   DATA[1809,37] := 189.2143;
   DATA[1809,38] := 0.000128152;
   DATA[1809,39] := 1.0;
   DATA[1809,40] := 1.0;
   DATA[1810,0] := 2.636198;
   DATA[1810,1] := 842.0502;
   DATA[1810,2] := 2.0;
   DATA[1810,3] := 1.0;
   DATA[1810,4] := 262.625;
   DATA[1810,5] := 8.46533;
   DATA[1810,6] := 320.0461;
   DATA[1810,8] := 1.0;
   DATA[1810,9] := 1.0;
   DATA[1810,10] := 1.0;
   DATA[1810,11] := 19.66835;
   DATA[1810,12] := 2.20645;
   DATA[1810,13] := 805.082;
   DATA[1810,14] := 1.0;
   DATA[1810,15] := 2.0;
   DATA[1810,16] := 1.0;
   DATA[1810,17] := 1.0;
   DATA[1810,18] := 1.0;
   DATA[1810,19] := 2.0;
   DATA[1810,20] := 148.808;
   DATA[1810,21] := 154.5501;
   DATA[1810,22] := 1.717746;
   DATA[1810,23] := 811.0997;
   DATA[1810,24] := 2.0;
   DATA[1810,25] := 2.0;
   DATA[1810,26] := 7.874455;
   DATA[1810,27] := 143.3222;
   DATA[1810,28] := 262.3686;
   DATA[1810,29] := 12.15073;
   DATA[1810,30] := 1.728019;
   DATA[1810,31] := 1.292174;
   DATA[1810,32] := 0.7351407;
   DATA[1810,33] := 0.306761;
   DATA[1810,34] := 2.0;
   DATA[1810,35] := 250.4005;
   DATA[1810,36] := 1.69801;
   DATA[1810,37] := 189.2143;
   DATA[1810,38] := 0.000128152;
   DATA[1810,39] := 1.0;
   DATA[1810,40] := 1.0;
   DATA[1811,0] := 2.65061;
   DATA[1811,1] := 842.6782;
   DATA[1811,2] := 2.0;
   DATA[1811,3] := 1.0;
   DATA[1811,4] := 262.625;
   DATA[1811,5] := 8.46533;
   DATA[1811,6] := 320.0461;
   DATA[1811,8] := 1.0;
   DATA[1811,9] := 1.0;
   DATA[1811,10] := 1.0;
   DATA[1811,11] := 19.72277;
   DATA[1811,12] := 2.20645;
   DATA[1811,13] := 804.5613;
   DATA[1811,14] := 1.0;
   DATA[1811,15] := 2.0;
   DATA[1811,16] := 1.0;
   DATA[1811,17] := 1.0;
   DATA[1811,18] := 1.0;
   DATA[1811,19] := 2.0;
   DATA[1811,20] := 148.808;
   DATA[1811,21] := 154.5501;
   DATA[1811,22] := 1.717746;
   DATA[1811,23] := 811.4843;
   DATA[1811,24] := 2.0;
   DATA[1811,25] := 2.0;
   DATA[1811,26] := 7.874455;
   DATA[1811,27] := 143.3222;
   DATA[1811,28] := 262.3686;
   DATA[1811,29] := 12.15073;
   DATA[1811,30] := 1.728147;
   DATA[1811,31] := 1.292174;
   DATA[1811,32] := 0.7351407;
   DATA[1811,33] := 0.3081703;
   DATA[1811,34] := 2.0;
   DATA[1811,35] := 250.4005;
   DATA[1811,36] := 1.69801;
   DATA[1811,37] := 189.2143;
   DATA[1811,38] := 0.000128152;
   DATA[1811,39] := 1.0;
   DATA[1811,40] := 1.0;
   DATA[1812,0] := 2.654133;
   DATA[1812,1] := 843.424;
   DATA[1812,2] := 2.0;
   DATA[1812,3] := 1.0;
   DATA[1812,4] := 262.625;
   DATA[1812,5] := 8.46533;
   DATA[1812,6] := 320.0461;
   DATA[1812,8] := 1.0;
   DATA[1812,9] := 1.0;
   DATA[1812,10] := 1.0;
   DATA[1812,11] := 19.72277;
   DATA[1812,12] := 2.209909;
   DATA[1812,13] := 803.9205;
   DATA[1812,14] := 1.0;
   DATA[1812,15] := 2.0;
   DATA[1812,16] := 1.0;
   DATA[1812,17] := 1.0;
   DATA[1812,18] := 1.0;
   DATA[1812,19] := 2.0;
   DATA[1812,20] := 148.808;
   DATA[1812,21] := 154.5501;
   DATA[1812,22] := 1.717746;
   DATA[1812,23] := 811.4843;
   DATA[1812,24] := 2.0;
   DATA[1812,25] := 2.0;
   DATA[1812,26] := 7.874455;
   DATA[1812,27] := 143.3222;
   DATA[1812,28] := 262.3686;
   DATA[1812,29] := 12.07383;
   DATA[1812,30] := 1.728147;
   DATA[1812,31] := 1.292174;
   DATA[1812,32] := 0.7351407;
   DATA[1812,33] := 0.3084905;
   DATA[1812,34] := 2.0;
   DATA[1812,35] := 250.4005;
   DATA[1812,36] := 1.69801;
   DATA[1812,37] := 189.2143;
   DATA[1812,38] := 0.000128152;
   DATA[1812,39] := 1.0;
   DATA[1812,40] := 1.0;
   DATA[1813,0] := 2.654133;
   DATA[1813,1] := 843.8558;
   DATA[1813,2] := 2.0;
   DATA[1813,3] := 1.0;
   DATA[1813,4] := 262.625;
   DATA[1813,5] := 8.46533;
   DATA[1813,6] := 320.0461;
   DATA[1813,8] := 1.0;
   DATA[1813,9] := 1.0;
   DATA[1813,10] := 1.0;
   DATA[1813,11] := 19.72277;
   DATA[1813,12] := 2.209909;
   DATA[1813,13] := 804.1207;
   DATA[1813,14] := 1.0;
   DATA[1813,15] := 2.0;
   DATA[1813,16] := 1.0;
   DATA[1813,17] := 1.0;
   DATA[1813,18] := 1.0;
   DATA[1813,19] := 2.0;
   DATA[1813,20] := 148.808;
   DATA[1813,21] := 154.5501;
   DATA[1813,22] := 1.717746;
   DATA[1813,23] := 812.0995;
   DATA[1813,24] := 2.0;
   DATA[1813,25] := 2.0;
   DATA[1813,26] := 7.874455;
   DATA[1813,27] := 143.3222;
   DATA[1813,28] := 262.3686;
   DATA[1813,29] := 12.07383;
   DATA[1813,30] := 1.727506;
   DATA[1813,31] := 1.281158;
   DATA[1813,32] := 0.7351407;
   DATA[1813,33] := 0.3084905;
   DATA[1813,34] := 2.0;
   DATA[1813,35] := 250.3365;
   DATA[1813,36] := 1.69801;
   DATA[1813,37] := 189.2143;
   DATA[1813,38] := 0.000128152;
   DATA[1813,39] := 1.0;
   DATA[1813,40] := 1.0;
   DATA[1814,0] := 2.628511;
   DATA[1814,1] := 844.7586;
   DATA[1814,2] := 2.0;
   DATA[1814,3] := 1.0;
   DATA[1814,4] := 262.625;
   DATA[1814,5] := 8.46533;
   DATA[1814,6] := 320.0461;
   DATA[1814,8] := 1.0;
   DATA[1814,9] := 1.0;
   DATA[1814,10] := 1.0;
   DATA[1814,11] := 19.69396;
   DATA[1814,12] := 2.209909;
   DATA[1814,13] := 803.3998;
   DATA[1814,14] := 1.0;
   DATA[1814,15] := 2.0;
   DATA[1814,16] := 1.0;
   DATA[1814,17] := 1.0;
   DATA[1814,18] := 1.0;
   DATA[1814,19] := 2.0;
   DATA[1814,20] := 148.808;
   DATA[1814,21] := 154.5501;
   DATA[1814,22] := 1.717746;
   DATA[1814,23] := 812.3302;
   DATA[1814,24] := 2.0;
   DATA[1814,25] := 2.0;
   DATA[1814,26] := 7.874455;
   DATA[1814,27] := 143.3222;
   DATA[1814,28] := 262.3686;
   DATA[1814,29] := 11.84312;
   DATA[1814,30] := 1.726737;
   DATA[1814,31] := 1.280646;
   DATA[1814,32] := 0.7351407;
   DATA[1814,33] := 0.3084905;
   DATA[1814,34] := 2.0;
   DATA[1814,35] := 250.2563;
   DATA[1814,36] := 1.69801;
   DATA[1814,37] := 189.022;
   DATA[1814,38] := 0.000128152;
   DATA[1814,39] := 1.0;
   DATA[1814,40] := 1.0;
   DATA[1815,0] := 2.620824;
   DATA[1815,1] := 844.9156;
   DATA[1815,2] := 2.0;
   DATA[1815,3] := 1.0;
   DATA[1815,4] := 262.625;
   DATA[1815,5] := 8.46533;
   DATA[1815,6] := 320.0461;
   DATA[1815,8] := 1.0;
   DATA[1815,9] := 1.0;
   DATA[1815,10] := 1.0;
   DATA[1815,11] := 19.69396;
   DATA[1815,12] := 2.209909;
   DATA[1815,13] := 802.5987;
   DATA[1815,14] := 1.0;
   DATA[1815,15] := 2.0;
   DATA[1815,16] := 1.0;
   DATA[1815,17] := 1.0;
   DATA[1815,18] := 1.0;
   DATA[1815,19] := 2.0;
   DATA[1815,20] := 148.808;
   DATA[1815,21] := 154.5501;
   DATA[1815,22] := 1.717746;
   DATA[1815,23] := 812.7531;
   DATA[1815,24] := 2.0;
   DATA[1815,25] := 2.0;
   DATA[1815,26] := 7.874455;
   DATA[1815,27] := 143.3222;
   DATA[1815,28] := 262.3686;
   DATA[1815,29] := 11.84312;
   DATA[1815,30] := 1.726737;
   DATA[1815,31] := 1.280646;
   DATA[1815,32] := 0.7351407;
   DATA[1815,33] := 0.3084905;
   DATA[1815,34] := 2.0;
   DATA[1815,35] := 250.1923;
   DATA[1815,36] := 1.69801;
   DATA[1815,37] := 189.022;
   DATA[1815,38] := 0.000128152;
   DATA[1815,39] := 1.0;
   DATA[1815,40] := 1.0;
   DATA[1816,0] := 2.606412;
   DATA[1816,1] := 845.5829;
   DATA[1816,2] := 2.0;
   DATA[1816,3] := 1.0;
   DATA[1816,4] := 262.625;
   DATA[1816,5] := 8.46533;
   DATA[1816,6] := 320.0461;
   DATA[1816,8] := 1.0;
   DATA[1816,9] := 1.0;
   DATA[1816,10] := 1.0;
   DATA[1816,11] := 19.73878;
   DATA[1816,12] := 2.209909;
   DATA[1816,13] := 801.9578;
   DATA[1816,14] := 1.0;
   DATA[1816,15] := 2.0;
   DATA[1816,16] := 1.0;
   DATA[1816,17] := 1.0;
   DATA[1816,18] := 1.0;
   DATA[1816,19] := 2.0;
   DATA[1816,20] := 148.808;
   DATA[1816,21] := 154.5501;
   DATA[1816,22] := 1.717746;
   DATA[1816,23] := 813.0223;
   DATA[1816,24] := 2.0;
   DATA[1816,25] := 2.0;
   DATA[1816,26] := 7.874455;
   DATA[1816,27] := 143.3222;
   DATA[1816,28] := 262.3686;
   DATA[1816,29] := 12.15073;
   DATA[1816,30] := 1.725455;
   DATA[1816,31] := 1.281927;
   DATA[1816,32] := 0.7357808;
   DATA[1816,33] := 0.3084905;
   DATA[1816,34] := 2.0;
   DATA[1816,35] := 250.1923;
   DATA[1816,36] := 1.69801;
   DATA[1816,37] := 189.022;
   DATA[1816,38] := 0.000128152;
   DATA[1816,39] := 1.0;
   DATA[1816,40] := 1.0;
   DATA[1817,0] := 2.593601;
   DATA[1817,1] := 846.0147;
   DATA[1817,2] := 2.0;
   DATA[1817,3] := 1.0;
   DATA[1817,4] := 262.625;
   DATA[1817,5] := 8.46533;
   DATA[1817,6] := 320.0461;
   DATA[1817,8] := 1.0;
   DATA[1817,9] := 1.0;
   DATA[1817,10] := 1.0;
   DATA[1817,11] := 19.74838;
   DATA[1817,12] := 2.209909;
   DATA[1817,13] := 801.1968;
   DATA[1817,14] := 1.0;
   DATA[1817,15] := 2.0;
   DATA[1817,16] := 1.0;
   DATA[1817,17] := 1.0;
   DATA[1817,18] := 1.0;
   DATA[1817,19] := 2.0;
   DATA[1817,20] := 148.808;
   DATA[1817,21] := 154.5501;
   DATA[1817,22] := 1.717746;
   DATA[1817,23] := 813.7144;
   DATA[1817,24] := 2.0;
   DATA[1817,25] := 2.0;
   DATA[1817,26] := 7.874455;
   DATA[1817,27] := 143.3222;
   DATA[1817,28] := 262.3686;
   DATA[1817,29] := 12.15073;
   DATA[1817,30] := 1.725455;
   DATA[1817,31] := 1.282439;
   DATA[1817,32] := 0.7357808;
   DATA[1817,33] := 0.3084905;
   DATA[1817,34] := 2.0;
   DATA[1817,35] := 250.1923;
   DATA[1817,36] := 1.69801;
   DATA[1817,37] := 189.022;
   DATA[1817,38] := 0.000128152;
   DATA[1817,39] := 1.0;
   DATA[1817,40] := 1.0;
   DATA[1818,0] := 2.5699;
   DATA[1818,1] := 846.682;
   DATA[1818,2] := 2.0;
   DATA[1818,3] := 1.0;
   DATA[1818,4] := 262.625;
   DATA[1818,5] := 8.46533;
   DATA[1818,6] := 320.0461;
   DATA[1818,8] := 1.0;
   DATA[1818,9] := 1.0;
   DATA[1818,10] := 1.0;
   DATA[1818,11] := 19.74838;
   DATA[1818,12] := 2.209909;
   DATA[1818,13] := 800.8764;
   DATA[1818,14] := 1.0;
   DATA[1818,15] := 2.0;
   DATA[1818,16] := 1.0;
   DATA[1818,17] := 1.0;
   DATA[1818,18] := 1.0;
   DATA[1818,19] := 2.0;
   DATA[1818,20] := 148.808;
   DATA[1818,21] := 154.5501;
   DATA[1818,22] := 1.717746;
   DATA[1818,23] := 813.5222;
   DATA[1818,24] := 2.0;
   DATA[1818,25] := 2.0;
   DATA[1818,26] := 7.874455;
   DATA[1818,27] := 143.3222;
   DATA[1818,28] := 262.3686;
   DATA[1818,29] := 12.15073;
   DATA[1818,30] := 1.725455;
   DATA[1818,31] := 1.282439;
   DATA[1818,32] := 0.7378293;
   DATA[1818,33] := 0.3084905;
   DATA[1818,34] := 2.0;
   DATA[1818,35] := 250.1923;
   DATA[1818,36] := 1.69801;
   DATA[1818,37] := 189.022;
   DATA[1818,38] := 0.000128152;
   DATA[1818,39] := 1.0;
   DATA[1818,40] := 1.0;
   DATA[1819,0] := 2.549723;
   DATA[1819,1] := 846.9568;
   DATA[1819,2] := 2.0;
   DATA[1819,3] := 1.0;
   DATA[1819,4] := 262.625;
   DATA[1819,5] := 8.46533;
   DATA[1819,6] := 320.0461;
   DATA[1819,8] := 1.0;
   DATA[1819,9] := 1.0;
   DATA[1819,10] := 1.0;
   DATA[1819,11] := 19.73238;
   DATA[1819,12] := 2.209909;
   DATA[1819,13] := 800.5159;
   DATA[1819,14] := 1.0;
   DATA[1819,15] := 2.0;
   DATA[1819,16] := 1.0;
   DATA[1819,17] := 1.0;
   DATA[1819,18] := 1.0;
   DATA[1819,19] := 2.0;
   DATA[1819,20] := 148.808;
   DATA[1819,21] := 154.5501;
   DATA[1819,22] := 1.715439;
   DATA[1819,23] := 813.676;
   DATA[1819,24] := 2.0;
   DATA[1819,25] := 2.0;
   DATA[1819,26] := 7.874455;
   DATA[1819,27] := 143.3222;
   DATA[1819,28] := 262.3686;
   DATA[1819,29] := 12.15073;
   DATA[1819,30] := 1.725455;
   DATA[1819,31] := 1.279877;
   DATA[1819,32] := 0.7387255;
   DATA[1819,33] := 0.3084905;
   DATA[1819,34] := 2.0;
   DATA[1819,35] := 250.1923;
   DATA[1819,36] := 1.69801;
   DATA[1819,37] := 189.022;
   DATA[1819,38] := 0.000128152;
   DATA[1819,39] := 1.0;
   DATA[1819,40] := 1.0;
   DATA[1820,0] := 2.528264;
   DATA[1820,1] := 847.7418;
   DATA[1820,2] := 2.0;
   DATA[1820,3] := 1.0;
   DATA[1820,4] := 262.625;
   DATA[1820,5] := 8.46533;
   DATA[1820,6] := 320.0461;
   DATA[1820,8] := 1.0;
   DATA[1820,9] := 1.0;
   DATA[1820,10] := 1.0;
   DATA[1820,11] := 19.68756;
   DATA[1820,12] := 2.208116;
   DATA[1820,13] := 800.1154;
   DATA[1820,14] := 1.0;
   DATA[1820,15] := 2.0;
   DATA[1820,16] := 1.0;
   DATA[1820,17] := 1.0;
   DATA[1820,18] := 1.0;
   DATA[1820,19] := 2.0;
   DATA[1820,20] := 148.808;
   DATA[1820,21] := 154.5501;
   DATA[1820,22] := 1.713901;
   DATA[1820,23] := 814.2912;
   DATA[1820,24] := 2.0;
   DATA[1820,25] := 2.0;
   DATA[1820,26] := 7.874455;
   DATA[1820,27] := 143.3222;
   DATA[1820,28] := 262.3686;
   DATA[1820,29] := 12.15073;
   DATA[1820,30] := 1.725455;
   DATA[1820,31] := 1.263994;
   DATA[1820,32] := 0.7357808;
   DATA[1820,33] := 0.3084905;
   DATA[1820,34] := 2.0;
   DATA[1820,35] := 250.0801;
   DATA[1820,36] := 1.69801;
   DATA[1820,37] := 189.022;
   DATA[1820,38] := 0.000128152;
   DATA[1820,39] := 1.0;
   DATA[1820,40] := 1.0;
   DATA[1821,0] := 2.516414;
   DATA[1821,1] := 848.1343;
   DATA[1821,2] := 2.0;
   DATA[1821,3] := 1.0;
   DATA[1821,4] := 262.625;
   DATA[1821,5] := 8.46533;
   DATA[1821,6] := 320.0461;
   DATA[1821,8] := 1.0;
   DATA[1821,9] := 1.0;
   DATA[1821,10] := 1.0;
   DATA[1821,11] := 19.68756;
   DATA[1821,12] := 2.208116;
   DATA[1821,13] := 799.7549;
   DATA[1821,14] := 1.0;
   DATA[1821,15] := 2.0;
   DATA[1821,16] := 1.0;
   DATA[1821,17] := 1.0;
   DATA[1821,18] := 1.0;
   DATA[1821,19] := 2.0;
   DATA[1821,20] := 148.808;
   DATA[1821,21] := 154.5501;
   DATA[1821,22] := 1.713645;
   DATA[1821,23] := 814.445;
   DATA[1821,24] := 2.0;
   DATA[1821,25] := 2.0;
   DATA[1821,26] := 7.874455;
   DATA[1821,27] := 143.3222;
   DATA[1821,28] := 262.3686;
   DATA[1821,29] := 12.15073;
   DATA[1821,30] := 1.724942;
   DATA[1821,31] := 1.261432;
   DATA[1821,32] := 0.7352687;
   DATA[1821,33] := 0.3084905;
   DATA[1821,34] := 2.0;
   DATA[1821,35] := 249.9519;
   DATA[1821,36] := 1.69801;
   DATA[1821,37] := 189.022;
   DATA[1821,38] := 0.000128152;
   DATA[1821,39] := 1.0;
   DATA[1821,40] := 1.0;
   DATA[1822,0] := 2.496877;
   DATA[1822,1] := 848.6839;
   DATA[1822,2] := 2.0;
   DATA[1822,3] := 1.0;
   DATA[1822,4] := 262.625;
   DATA[1822,5] := 8.46533;
   DATA[1822,6] := 320.0461;
   DATA[1822,9] := 1.0;
   DATA[1822,10] := 1.0;
   DATA[1822,11] := 19.72598;
   DATA[1822,12] := 2.208116;
   DATA[1822,13] := 799.3143;
   DATA[1822,14] := 1.0;
   DATA[1822,15] := 2.0;
   DATA[1822,16] := 1.0;
   DATA[1822,17] := 1.0;
   DATA[1822,18] := 1.0;
   DATA[1822,19] := 2.0;
   DATA[1822,20] := 148.808;
   DATA[1822,21] := 154.5501;
   DATA[1822,22] := 1.712363;
   DATA[1822,23] := 814.8295;
   DATA[1822,24] := 2.0;
   DATA[1822,25] := 2.0;
   DATA[1822,26] := 7.874455;
   DATA[1822,27] := 143.3222;
   DATA[1822,28] := 262.3686;
   DATA[1822,29] := 12.15073;
   DATA[1822,30] := 1.724045;
   DATA[1822,31] := 1.261432;
   DATA[1822,32] := 0.7348846;
   DATA[1822,33] := 0.3084905;
   DATA[1822,34] := 2.0;
   DATA[1822,35] := 249.9519;
   DATA[1822,36] := 1.69801;
   DATA[1822,37] := 189.022;
   DATA[1822,38] := 0.000128152;
   DATA[1822,39] := 1.0;
   DATA[1822,40] := 1.0;
   DATA[1823,0] := 2.481504;
   DATA[1823,1] := 849.5082;
   DATA[1823,2] := 2.0;
   DATA[1823,3] := 1.0;
   DATA[1823,4] := 262.625;
   DATA[1823,5] := 8.46533;
   DATA[1823,6] := 320.0461;
   DATA[1823,9] := 1.0;
   DATA[1823,10] := 1.0;
   DATA[1823,11] := 19.75159;
   DATA[1823,12] := 2.209653;
   DATA[1823,13] := 799.1541;
   DATA[1823,14] := 1.0;
   DATA[1823,15] := 2.0;
   DATA[1823,16] := 1.0;
   DATA[1823,17] := 1.0;
   DATA[1823,18] := 1.0;
   DATA[1823,19] := 2.0;
   DATA[1823,20] := 148.808;
   DATA[1823,21] := 154.5501;
   DATA[1823,22] := 1.712363;
   DATA[1823,23] := 814.8295;
   DATA[1823,24] := 2.0;
   DATA[1823,25] := 2.0;
   DATA[1823,26] := 7.874455;
   DATA[1823,27] := 143.3222;
   DATA[1823,28] := 262.3686;
   DATA[1823,29] := 12.15073;
   DATA[1823,30] := 1.723532;
   DATA[1823,31] := 1.261432;
   DATA[1823,32] := 0.7355248;
   DATA[1823,33] := 0.3084905;
   DATA[1823,34] := 2.0;
   DATA[1823,35] := 249.9519;
   DATA[1823,36] := 1.69801;
   DATA[1823,37] := 188.9259;
   DATA[1823,38] := 0.000128152;
   DATA[1823,39] := 1.0;
   DATA[1823,40] := 1.0;
   DATA[1824,0] := 2.461006;
   DATA[1824,1] := 849.8222;
   DATA[1824,2] := 2.0;
   DATA[1824,3] := 1.0;
   DATA[1824,4] := 262.625;
   DATA[1824,5] := 8.46533;
   DATA[1824,6] := 320.2;
   DATA[1824,9] := 1.0;
   DATA[1824,10] := 1.0;
   DATA[1824,11] := 19.75159;
   DATA[1824,12] := 2.209653;
   DATA[1824,13] := 798.9138;
   DATA[1824,14] := 1.0;
   DATA[1824,15] := 2.0;
   DATA[1824,16] := 1.0;
   DATA[1824,17] := 1.0;
   DATA[1824,18] := 1.0;
   DATA[1824,19] := 2.0;
   DATA[1824,20] := 148.808;
   DATA[1824,21] := 154.5501;
   DATA[1824,22] := 1.712363;
   DATA[1824,23] := 815.3294;
   DATA[1824,24] := 2.0;
   DATA[1824,25] := 2.0;
   DATA[1824,26] := 7.874455;
   DATA[1824,27] := 143.3222;
   DATA[1824,28] := 262.3686;
   DATA[1824,29] := 12.15073;
   DATA[1824,30] := 1.723532;
   DATA[1824,31] := 1.272192;
   DATA[1824,32] := 0.7377012;
   DATA[1824,33] := 0.3084905;
   DATA[1824,34] := 2.0;
   DATA[1824,35] := 249.9519;
   DATA[1824,36] := 1.69801;
   DATA[1824,37] := 188.9259;
   DATA[1824,38] := 0.000128152;
   DATA[1824,39] := 1.0;
   DATA[1824,40] := 1.0;
   DATA[1825,0] := 2.449156;
   DATA[1825,1] := 850.8035;
   DATA[1825,2] := 2.0;
   DATA[1825,3] := 1.0;
   DATA[1825,4] := 262.625;
   DATA[1825,5] := 8.46533;
   DATA[1825,6] := 320.2;
   DATA[1825,9] := 1.0;
   DATA[1825,10] := 1.0;
   DATA[1825,11] := 19.75159;
   DATA[1825,12] := 2.209653;
   DATA[1825,13] := 798.5933;
   DATA[1825,14] := 1.0;
   DATA[1825,15] := 2.0;
   DATA[1825,16] := 1.0;
   DATA[1825,17] := 1.0;
   DATA[1825,18] := 1.0;
   DATA[1825,19] := 2.0;
   DATA[1825,20] := 148.808;
   DATA[1825,21] := 154.5501;
   DATA[1825,22] := 1.712363;
   DATA[1825,23] := 815.5217;
   DATA[1825,24] := 2.0;
   DATA[1825,25] := 2.0;
   DATA[1825,26] := 7.874455;
   DATA[1825,27] := 143.3222;
   DATA[1825,28] := 262.3686;
   DATA[1825,29] := 12.15073;
   DATA[1825,30] := 1.723532;
   DATA[1825,31] := 1.272192;
   DATA[1825,32] := 0.7377012;
   DATA[1825,33] := 0.3084905;
   DATA[1825,34] := 2.0;
   DATA[1825,35] := 249.9519;
   DATA[1825,36] := 1.69801;
   DATA[1825,37] := 188.9259;
   DATA[1825,38] := 0.000128152;
   DATA[1825,39] := 1.0;
   DATA[1825,40] := 1.0;
   DATA[1826,0] := 2.433462;
   DATA[1826,1] := 851.0391;
   DATA[1826,2] := 2.0;
   DATA[1826,3] := 1.0;
   DATA[1826,4] := 262.625;
   DATA[1826,5] := 8.46533;
   DATA[1826,6] := 320.2;
   DATA[1826,9] := 1.0;
   DATA[1826,10] := 1.0;
   DATA[1826,11] := 19.7996;
   DATA[1826,12] := 2.209653;
   DATA[1826,13] := 798.353;
   DATA[1826,14] := 1.0;
   DATA[1826,15] := 2.0;
   DATA[1826,16] := 1.0;
   DATA[1826,17] := 1.0;
   DATA[1826,18] := 1.0;
   DATA[1826,19] := 2.0;
   DATA[1826,20] := 148.808;
   DATA[1826,21] := 154.5501;
   DATA[1826,22] := 1.712363;
   DATA[1826,23] := 815.5986;
   DATA[1826,24] := 2.0;
   DATA[1826,25] := 2.0;
   DATA[1826,26] := 7.874455;
   DATA[1826,27] := 143.3222;
   DATA[1826,28] := 262.3686;
   DATA[1826,29] := 12.15073;
   DATA[1826,30] := 1.723532;
   DATA[1826,31] := 1.272192;
   DATA[1826,32] := 0.7348846;
   DATA[1826,33] := 0.3084905;
   DATA[1826,34] := 2.0;
   DATA[1826,35] := 249.9519;
   DATA[1826,36] := 1.585878;
   DATA[1826,37] := 188.9259;
   DATA[1826,38] := 0.000128152;
   DATA[1826,39] := 1.0;
   DATA[1826,40] := 1.0;
   DATA[1827,0] := 2.433462;
   DATA[1827,1] := 851.0391;
   DATA[1827,2] := 2.0;
   DATA[1827,3] := 1.0;
   DATA[1827,4] := 262.625;
   DATA[1827,5] := 8.46533;
   DATA[1827,6] := 320.2;
   DATA[1827,9] := 1.0;
   DATA[1827,10] := 1.0;
   DATA[1827,11] := 19.7996;
   DATA[1827,12] := 2.209653;
   DATA[1827,13] := 798.353;
   DATA[1827,14] := 1.0;
   DATA[1827,15] := 2.0;
   DATA[1827,16] := 1.0;
   DATA[1827,17] := 1.0;
   DATA[1827,18] := 1.0;
   DATA[1827,19] := 2.0;
   DATA[1827,20] := 148.808;
   DATA[1827,21] := 154.5501;
   DATA[1827,22] := 1.712363;
   DATA[1827,23] := 815.5986;
   DATA[1827,24] := 2.0;
   DATA[1827,25] := 2.0;
   DATA[1827,26] := 7.874455;
   DATA[1827,27] := 143.3222;
   DATA[1827,28] := 262.3686;
   DATA[1827,29] := 12.15073;
   DATA[1827,30] := 1.723532;
   DATA[1827,31] := 1.272192;
   DATA[1827,32] := 0.7348846;
   DATA[1827,33] := 0.3084905;
   DATA[1827,34] := 2.0;
   DATA[1827,35] := 249.9519;
   DATA[1827,36] := 1.585878;
   DATA[1827,37] := 188.9259;
   DATA[1827,38] := 0.000128152;
   DATA[1827,39] := 1.0;
   DATA[1827,40] := 1.0;
   DATA[1828,0] := 2.427057;
   DATA[1828,1] := 851.5101;
   DATA[1828,2] := 2.0;
   DATA[1828,3] := 1.0;
   DATA[1828,4] := 262.625;
   DATA[1828,5] := 8.46533;
   DATA[1828,6] := 320.2;
   DATA[1828,9] := 1.0;
   DATA[1828,10] := 1.0;
   DATA[1828,11] := 19.7996;
   DATA[1828,12] := 2.209653;
   DATA[1828,13] := 797.7522;
   DATA[1828,14] := 1.0;
   DATA[1828,15] := 2.0;
   DATA[1828,16] := 1.0;
   DATA[1828,17] := 1.0;
   DATA[1828,18] := 1.0;
   DATA[1828,19] := 2.0;
   DATA[1828,20] := 148.808;
   DATA[1828,21] := 154.5501;
   DATA[1828,22] := 1.712363;
   DATA[1828,23] := 815.7908;
   DATA[1828,24] := 2.0;
   DATA[1828,25] := 2.0;
   DATA[1828,26] := 7.874455;
   DATA[1828,27] := 143.3222;
   DATA[1828,28] := 262.3686;
   DATA[1828,29] := 12.15073;
   DATA[1828,30] := 1.723532;
   DATA[1828,31] := 1.266428;
   DATA[1828,32] := 0.7348846;
   DATA[1828,33] := 0.3084905;
   DATA[1828,34] := 2.0;
   DATA[1828,35] := 250.0;
   DATA[1828,36] := 1.585878;
   DATA[1828,37] := 188.9259;
   DATA[1828,38] := 0.000128152;
   DATA[1828,39] := 1.0;
   DATA[1828,40] := 1.0;
   DATA[1829,0] := 2.427057;
   DATA[1829,1] := 851.9811;
   DATA[1829,2] := 2.0;
   DATA[1829,3] := 1.0;
   DATA[1829,4] := 262.625;
   DATA[1829,5] := 8.46533;
   DATA[1829,6] := 320.2;
   DATA[1829,9] := 1.0;
   DATA[1829,10] := 1.0;
   DATA[1829,11] := 19.73238;
   DATA[1829,12] := 2.209653;
   DATA[1829,13] := 797.4718;
   DATA[1829,14] := 1.0;
   DATA[1829,15] := 2.0;
   DATA[1829,16] := 1.0;
   DATA[1829,17] := 1.0;
   DATA[1829,18] := 1.0;
   DATA[1829,19] := 2.0;
   DATA[1829,20] := 148.808;
   DATA[1829,21] := 154.5501;
   DATA[1829,22] := 1.712363;
   DATA[1829,23] := 816.1754;
   DATA[1829,24] := 2.0;
   DATA[1829,25] := 2.0;
   DATA[1829,26] := 7.874455;
   DATA[1829,27] := 143.3222;
   DATA[1829,28] := 262.3686;
   DATA[1829,29] := 12.15073;
   DATA[1829,30] := 1.723532;
   DATA[1829,31] := 1.261944;
   DATA[1829,32] := 0.7348846;
   DATA[1829,33] := 0.3084905;
   DATA[1829,34] := 2.0;
   DATA[1829,35] := 250.0;
   DATA[1829,36] := 1.585878;
   DATA[1829,37] := 188.9259;
   DATA[1829,38] := 0.000128152;
   DATA[1829,39] := 1.0;
   DATA[1829,40] := 1.0;
   DATA[1830,0] := 2.438267;
   DATA[1830,1] := 852.7662;
   DATA[1830,2] := 2.0;
   DATA[1830,3] := 1.0;
   DATA[1830,4] := 262.625;
   DATA[1830,5] := 8.46533;
   DATA[1830,6] := 319.9949;
   DATA[1830,9] := 1.0;
   DATA[1830,10] := 1.0;
   DATA[1830,11] := 19.70997;
   DATA[1830,12] := 2.207731;
   DATA[1830,13] := 797.2715;
   DATA[1830,14] := 1.0;
   DATA[1830,15] := 2.0;
   DATA[1830,16] := 1.0;
   DATA[1830,17] := 1.0;
   DATA[1830,18] := 1.0;
   DATA[1830,19] := 2.0;
   DATA[1830,20] := 148.808;
   DATA[1830,21] := 154.5501;
   DATA[1830,22] := 1.712363;
   DATA[1830,23] := 816.3292;
   DATA[1830,24] := 2.0;
   DATA[1830,25] := 2.0;
   DATA[1830,26] := 7.874455;
   DATA[1830,27] := 143.3222;
   DATA[1830,28] := 262.3686;
   DATA[1830,29] := 12.15073;
   DATA[1830,30] := 1.723532;
   DATA[1830,31] := 1.261432;
   DATA[1830,32] := 0.7348846;
   DATA[1830,33] := 0.3084905;
   DATA[1830,34] := 2.0;
   DATA[1830,35] := 250.0;
   DATA[1830,36] := 1.649953;
   DATA[1830,37] := 188.8138;
   DATA[1830,38] := 0.000128152;
   DATA[1830,39] := 1.0;
   DATA[1830,40] := 1.0;
   DATA[1831,0] := 2.480223;
   DATA[1831,1] := 853.0802;
   DATA[1831,2] := 2.0;
   DATA[1831,3] := 2.0;
   DATA[1831,4] := 262.625;
   DATA[1831,5] := 8.46533;
   DATA[1831,6] := 319.9949;
   DATA[1831,8] := 2.0;
   DATA[1831,9] := 1.0;
   DATA[1831,10] := 1.0;
   DATA[1831,11] := 19.70037;
   DATA[1831,12] := 2.206835;
   DATA[1831,13] := 796.9911;
   DATA[1831,14] := 1.0;
   DATA[1831,15] := 2.0;
   DATA[1831,16] := 1.0;
   DATA[1831,17] := 1.0;
   DATA[1831,18] := 1.0;
   DATA[1831,19] := 2.0;
   DATA[1831,20] := 148.808;
   DATA[1831,21] := 154.5501;
   DATA[1831,22] := 1.712876;
   DATA[1831,23] := 816.3676;
   DATA[1831,24] := 2.0;
   DATA[1831,25] := 2.0;
   DATA[1831,26] := 7.874455;
   DATA[1831,27] := 143.3222;
   DATA[1831,28] := 262.3686;
   DATA[1831,29] := 12.15073;
   DATA[1831,30] := 1.723532;
   DATA[1831,31] := 1.261432;
   DATA[1831,32] := 0.7348846;
   DATA[1831,33] := 0.3084905;
   DATA[1831,34] := 2.0;
   DATA[1831,35] := 250.0;
   DATA[1831,36] := 1.649953;
   DATA[1831,37] := 188.8138;
   DATA[1831,38] := 0.000128152;
   DATA[1831,39] := 1.0;
   DATA[1831,40] := 1.0;
   DATA[1832,0] := 2.524101;
   DATA[1832,1] := 854.3363;
   DATA[1832,2] := 2.0;
   DATA[1832,3] := 2.0;
   DATA[1832,4] := 262.625;
   DATA[1832,5] := 8.46533;
   DATA[1832,6] := 319.9949;
   DATA[1832,8] := 2.0;
   DATA[1832,9] := 1.0;
   DATA[1832,10] := 1.0;
   DATA[1832,11] := 19.70037;
   DATA[1832,12] := 2.206835;
   DATA[1832,13] := 796.7909;
   DATA[1832,14] := 1.0;
   DATA[1832,15] := 2.0;
   DATA[1832,16] := 1.0;
   DATA[1832,17] := 1.0;
   DATA[1832,18] := 1.0;
   DATA[1832,19] := 2.0;
   DATA[1832,20] := 148.808;
   DATA[1832,21] := 154.5501;
   DATA[1832,22] := 1.713004;
   DATA[1832,23] := 816.3292;
   DATA[1832,24] := 2.0;
   DATA[1832,25] := 2.0;
   DATA[1832,26] := 7.874455;
   DATA[1832,27] := 143.3735;
   DATA[1832,28] := 262.3686;
   DATA[1832,29] := 12.15073;
   DATA[1832,30] := 1.723532;
   DATA[1832,31] := 1.270783;
   DATA[1832,32] := 0.7348846;
   DATA[1832,33] := 0.3084905;
   DATA[1832,34] := 2.0;
   DATA[1832,35] := 250.0;
   DATA[1832,36] := 1.649953;
   DATA[1832,37] := 188.8138;
   DATA[1832,38] := 0.000128152;
   DATA[1832,39] := 1.0;
   DATA[1832,40] := 1.0;
   DATA[1833,0] := 2.563174;
   DATA[1833,1] := 855.0036;
   DATA[1833,2] := 2.0;
   DATA[1833,3] := 2.0;
   DATA[1833,4] := 262.625;
   DATA[1833,5] := 8.46533;
   DATA[1833,6] := 319.9949;
   DATA[1833,7] := 0.02037613;
   DATA[1833,8] := 2.0;
   DATA[1833,9] := 1.0;
   DATA[1833,10] := 1.0;
   DATA[1833,11] := 19.70037;
   DATA[1833,12] := 2.206835;
   DATA[1833,13] := 796.3904;
   DATA[1833,14] := 1.0;
   DATA[1833,15] := 2.0;
   DATA[1833,16] := 1.0;
   DATA[1833,17] := 1.0;
   DATA[1833,18] := 1.0;
   DATA[1833,19] := 2.0;
   DATA[1833,20] := 148.808;
   DATA[1833,21] := 154.4219;
   DATA[1833,22] := 1.713004;
   DATA[1833,23] := 816.3292;
   DATA[1833,24] := 2.0;
   DATA[1833,25] := 2.0;
   DATA[1833,26] := 7.874455;
   DATA[1833,27] := 143.3735;
   DATA[1833,28] := 262.3686;
   DATA[1833,29] := 12.15073;
   DATA[1833,30] := 1.723532;
   DATA[1833,31] := 1.286153;
   DATA[1833,32] := 0.7355248;
   DATA[1833,33] := 0.3084905;
   DATA[1833,34] := 2.0;
   DATA[1833,35] := 250.0;
   DATA[1833,36] := 1.649953;
   DATA[1833,37] := 188.8138;
   DATA[1833,38] := 0.000128152;
   DATA[1833,39] := 1.0;
   DATA[1833,40] := 1.0;
   DATA[1834,0] := 2.60417;
   DATA[1834,1] := 855.5531;
   DATA[1834,2] := 2.0;
   DATA[1834,3] := 2.0;
   DATA[1834,4] := 262.625;
   DATA[1834,5] := 8.46533;
   DATA[1834,6] := 319.9949;
   DATA[1834,7] := 0.1724922;
   DATA[1834,8] := 2.0;
   DATA[1834,9] := 1.0;
   DATA[1834,10] := 1.0;
   DATA[1834,11] := 19.70037;
   DATA[1834,12] := 2.206835;
   DATA[1834,13] := 795.7095;
   DATA[1834,14] := 1.0;
   DATA[1834,15] := 2.0;
   DATA[1834,16] := 1.0;
   DATA[1834,17] := 1.0;
   DATA[1834,18] := 1.0;
   DATA[1834,19] := 2.0;
   DATA[1834,20] := 148.808;
   DATA[1834,21] := 154.4219;
   DATA[1834,22] := 1.713004;
   DATA[1834,23] := 816.5214;
   DATA[1834,24] := 2.0;
   DATA[1834,25] := 2.0;
   DATA[1834,26] := 7.874455;
   DATA[1834,27] := 143.3735;
   DATA[1834,28] := 262.3686;
   DATA[1834,29] := 12.15073;
   DATA[1834,30] := 1.723532;
   DATA[1834,31] := 1.289228;
   DATA[1834,32] := 0.7355248;
   DATA[1834,33] := 0.3084905;
   DATA[1834,34] := 2.0;
   DATA[1834,35] := 250.0;
   DATA[1834,36] := 1.649953;
   DATA[1834,37] := 188.8138;
   DATA[1834,38] := 0.000128152;
   DATA[1834,39] := 1.0;
   DATA[1834,40] := 1.0;
   DATA[1835,0] := 2.628511;
   DATA[1835,1] := 855.8279;
   DATA[1835,2] := 2.0;
   DATA[1835,3] := 2.0;
   DATA[1835,4] := 262.625;
   DATA[1835,5] := 8.46533;
   DATA[1835,6] := 319.9949;
   DATA[1835,7] := 0.4093166;
   DATA[1835,8] := 2.0;
   DATA[1835,9] := 1.0;
   DATA[1835,10] := 1.0;
   DATA[1835,11] := 19.70037;
   DATA[1835,12] := 2.206835;
   DATA[1835,13] := 795.1888;
   DATA[1835,14] := 1.0;
   DATA[1835,15] := 2.0;
   DATA[1835,16] := 1.0;
   DATA[1835,17] := 1.0;
   DATA[1835,18] := 1.0;
   DATA[1835,19] := 2.0;
   DATA[1835,20] := 148.808;
   DATA[1835,21] := 154.4219;
   DATA[1835,22] := 1.713004;
   DATA[1835,23] := 816.4061;
   DATA[1835,24] := 2.0;
   DATA[1835,25] := 2.0;
   DATA[1835,26] := 7.874135;
   DATA[1835,27] := 143.3735;
   DATA[1835,28] := 262.3686;
   DATA[1835,29] := 12.15073;
   DATA[1835,30] := 1.724686;
   DATA[1835,31] := 1.282311;
   DATA[1835,32] := 0.7355248;
   DATA[1835,33] := 0.3084905;
   DATA[1835,34] := 2.0;
   DATA[1835,35] := 250.0;
   DATA[1835,36] := 1.826162;
   DATA[1835,37] := 188.8138;
   DATA[1835,38] := 0.000128152;
   DATA[1835,39] := 1.0;
   DATA[1835,40] := 1.0;
   DATA[1836,0] := 2.654774;
   DATA[1836,1] := 856.77;
   DATA[1836,2] := 2.0;
   DATA[1836,3] := 2.0;
   DATA[1836,4] := 263.9067;
   DATA[1836,5] := 8.46533;
   DATA[1836,6] := 320.2;
   DATA[1836,7] := 0.7616057;
   DATA[1836,8] := 2.0;
   DATA[1836,9] := 1.0;
   DATA[1836,10] := 1.0;
   DATA[1836,11] := 19.70037;
   DATA[1836,12] := 2.210037;
   DATA[1836,13] := 794.3076;
   DATA[1836,14] := 1.0;
   DATA[1836,15] := 2.0;
   DATA[1836,16] := 1.0;
   DATA[1836,17] := 1.0;
   DATA[1836,18] := 1.0;
   DATA[1836,19] := 2.0;
   DATA[1836,20] := 148.808;
   DATA[1836,21] := 154.3707;
   DATA[1836,22] := 1.714926;
   DATA[1836,23] := 816.2907;
   DATA[1836,24] := 2.0;
   DATA[1836,25] := 2.0;
   DATA[1836,26] := 7.874135;
   DATA[1836,27] := 143.7324;
   DATA[1836,28] := 262.3686;
   DATA[1836,29] := 11.88157;
   DATA[1836,30] := 1.724686;
   DATA[1836,31] := 1.281158;
   DATA[1836,32] := 0.7355248;
   DATA[1836,33] := 0.3084905;
   DATA[1836,34] := 2.0;
   DATA[1836,35] := 249.8238;
   DATA[1836,36] := 1.826162;
   DATA[1836,37] := 188.7657;
   DATA[1836,38] := 0.000128152;
   DATA[1836,39] := 1.0;
   DATA[1836,40] := 1.0;
   DATA[1837,0] := 2.660859;
   DATA[1837,1] := 857.1232;
   DATA[1837,2] := 2.0;
   DATA[1837,3] := 2.0;
   DATA[1837,4] := 264.4194;
   DATA[1837,5] := 8.46533;
   DATA[1837,6] := 320.7639;
   DATA[1837,7] := 1.252683;
   DATA[1837,8] := 2.0;
   DATA[1837,9] := 1.0;
   DATA[1837,10] := 1.0;
   DATA[1837,11] := 19.70997;
   DATA[1837,12] := 2.210037;
   DATA[1837,13] := 793.7068;
   DATA[1837,14] := 1.0;
   DATA[1837,15] := 2.0;
   DATA[1837,16] := 1.0;
   DATA[1837,17] := 1.0;
   DATA[1837,18] := 1.0;
   DATA[1837,19] := 2.0;
   DATA[1837,20] := 148.808;
   DATA[1837,21] := 154.3707;
   DATA[1837,22] := 1.714542;
   DATA[1837,23] := 815.9062;
   DATA[1837,24] := 2.0;
   DATA[1837,25] := 2.0;
   DATA[1837,26] := 7.874135;
   DATA[1837,27] := 143.7324;
   DATA[1837,28] := 262.3686;
   DATA[1837,29] := 11.88157;
   DATA[1837,30] := 1.724686;
   DATA[1837,31] := 1.281158;
   DATA[1837,32] := 0.7355248;
   DATA[1837,33] := 0.3084905;
   DATA[1837,34] := 2.0;
   DATA[1837,35] := 249.7597;
   DATA[1837,36] := 1.826162;
   DATA[1837,37] := 188.6055;
   DATA[1837,38] := 0.000128152;
   DATA[1837,39] := 1.0;
   DATA[1837,40] := 1.0;
   DATA[1838,0] := 2.652532;
   DATA[1838,1] := 857.6728;
   DATA[1838,2] := 2.0;
   DATA[1838,3] := 2.0;
   DATA[1838,4] := 264.4194;
   DATA[1838,5] := 8.46533;
   DATA[1838,6] := 320.969;
   DATA[1838,7] := 1.414539;
   DATA[1838,8] := 2.0;
   DATA[1838,9] := 1.0;
   DATA[1838,10] := 1.0;
   DATA[1838,11] := 19.70997;
   DATA[1838,12] := 2.210037;
   DATA[1838,13] := 793.5065;
   DATA[1838,14] := 1.0;
   DATA[1838,15] := 2.0;
   DATA[1838,16] := 1.0;
   DATA[1838,17] := 1.0;
   DATA[1838,18] := 1.0;
   DATA[1838,19] := 2.0;
   DATA[1838,20] := 148.808;
   DATA[1838,21] := 154.3707;
   DATA[1838,22] := 1.713389;
   DATA[1838,23] := 815.5601;
   DATA[1838,24] := 2.0;
   DATA[1838,25] := 2.0;
   DATA[1838,26] := 7.874135;
   DATA[1838,27] := 143.4504;
   DATA[1838,28] := 262.3686;
   DATA[1838,29] := 11.88157;
   DATA[1838,30] := 1.724686;
   DATA[1838,31] := 1.281158;
   DATA[1838,32] := 0.7355248;
   DATA[1838,33] := 0.3084905;
   DATA[1838,34] := 2.0;
   DATA[1838,35] := 249.7597;
   DATA[1838,36] := 1.778105;
   DATA[1838,37] := 188.6055;
   DATA[1838,38] := 0.000128152;
   DATA[1838,39] := 1.0;
   DATA[1838,40] := 1.0;
   DATA[1839,0] := 2.641322;
   DATA[1839,1] := 857.9475;
   DATA[1839,2] := 2.0;
   DATA[1839,3] := 2.0;
   DATA[1839,4] := 264.4194;
   DATA[1839,5] := 8.464048;
   DATA[1839,6] := 321.6098;
   DATA[1839,7] := 1.852177;
   DATA[1839,8] := 2.0;
   DATA[1839,9] := 1.0;
   DATA[1839,10] := 1.0;
   DATA[1839,11] := 19.70997;
   DATA[1839,12] := 2.209013;
   DATA[1839,13] := 793.3062;
   DATA[1839,14] := 1.0;
   DATA[1839,15] := 2.0;
   DATA[1839,16] := 1.0;
   DATA[1839,17] := 1.0;
   DATA[1839,18] := 1.0;
   DATA[1839,19] := 2.0;
   DATA[1839,20] := 148.808;
   DATA[1839,21] := 154.3707;
   DATA[1839,22] := 1.711466;
   DATA[1839,23] := 815.9831;
   DATA[1839,24] := 2.0;
   DATA[1839,25] := 2.0;
   DATA[1839,26] := 7.874135;
   DATA[1839,27] := 143.4504;
   DATA[1839,28] := 262.3686;
   DATA[1839,29] := 11.88157;
   DATA[1839,30] := 1.724045;
   DATA[1839,31] := 1.285129;
   DATA[1839,32] := 0.7355248;
   DATA[1839,33] := 0.3084905;
   DATA[1839,34] := 2.0;
   DATA[1839,35] := 249.6315;
   DATA[1839,36] := 1.778105;
   DATA[1839,37] := 188.6055;
   DATA[1839,38] := 0.000128152;
   DATA[1839,39] := 1.0;
   DATA[1839,40] := 1.0;
   DATA[1840,0] := 2.625949;
   DATA[1840,1] := 858.3793;
   DATA[1840,2] := 2.0;
   DATA[1840,3] := 2.0;
   DATA[1840,4] := 264.4194;
   DATA[1840,5] := 8.460203;
   DATA[1840,6] := 322.3532;
   DATA[1840,7] := 2.185115;
   DATA[1840,8] := 2.0;
   DATA[1840,9] := 2.0;
   DATA[1840,10] := 2.0;
   DATA[1840,11] := 19.64594;
   DATA[1840,12] := 2.207347;
   DATA[1840,13] := 792.7855;
   DATA[1840,14] := 1.0;
   DATA[1840,15] := 2.0;
   DATA[1840,16] := 1.0;
   DATA[1840,17] := 1.0;
   DATA[1840,18] := 1.0;
   DATA[1840,19] := 2.0;
   DATA[1840,20] := 148.808;
   DATA[1840,21] := 154.3707;
   DATA[1840,22] := 1.711466;
   DATA[1840,23] := 815.8293;
   DATA[1840,24] := 2.0;
   DATA[1840,25] := 2.0;
   DATA[1840,26] := 7.874135;
   DATA[1840,27] := 143.4504;
   DATA[1840,28] := 262.3686;
   DATA[1840,29] := 11.88157;
   DATA[1840,30] := 1.722123;
   DATA[1840,31] := 1.296913;
   DATA[1840,32] := 0.7355248;
   DATA[1840,33] := 0.3084905;
   DATA[1840,34] := 2.0;
   DATA[1840,35] := 249.6315;
   DATA[1840,36] := 1.778105;
   DATA[1840,37] := 188.6055;
   DATA[1840,38] := 0.000128152;
   DATA[1840,39] := 1.0;
   DATA[1840,40] := 1.0;
   DATA[1841,0] := 2.621145;
   DATA[1841,1] := 858.6934;
   DATA[1841,2] := 2.0;
   DATA[1841,3] := 2.0;
   DATA[1841,4] := 264.4194;
   DATA[1841,5] := 8.458601;
   DATA[1841,6] := 323.1223;
   DATA[1841,7] := 2.298401;
   DATA[1841,8] := 2.0;
   DATA[1841,9] := 2.0;
   DATA[1841,10] := 2.0;
   DATA[1841,11] := 19.64594;
   DATA[1841,12] := 2.206963;
   DATA[1841,13] := 792.0646;
   DATA[1841,14] := 1.0;
   DATA[1841,15] := 2.0;
   DATA[1841,16] := 1.0;
   DATA[1841,17] := 1.0;
   DATA[1841,18] := 1.0;
   DATA[1841,19] := 2.0;
   DATA[1841,20] := 148.808;
   DATA[1841,21] := 154.3707;
   DATA[1841,22] := 1.713004;
   DATA[1841,23] := 815.7139;
   DATA[1841,24] := 2.0;
   DATA[1841,25] := 2.0;
   DATA[1841,26] := 7.874135;
   DATA[1841,27] := 143.4504;
   DATA[1841,28] := 262.3686;
   DATA[1841,29] := 11.88157;
   DATA[1841,30] := 1.722123;
   DATA[1841,31] := 1.30178;
   DATA[1841,32] := 0.7355248;
   DATA[1841,33] := 0.3084905;
   DATA[1841,34] := 2.0;
   DATA[1841,35] := 249.7917;
   DATA[1841,36] := 1.69801;
   DATA[1841,37] := 188.6055;
   DATA[1841,38] := 0.000128152;
   DATA[1841,39] := 1.0;
   DATA[1841,40] := 1.0;
   DATA[1842,0] := 2.609615;
   DATA[1842,1] := 858.8896;
   DATA[1842,2] := 2.0;
   DATA[1842,3] := 2.0;
   DATA[1842,4] := 264.4194;
   DATA[1842,5] := 8.451231;
   DATA[1842,6] := 324.3271;
   DATA[1842,7] := 2.373242;
   DATA[1842,8] := 2.0;
   DATA[1842,9] := 2.0;
   DATA[1842,10] := 2.0;
   DATA[1842,11] := 19.69076;
   DATA[1842,12] := 2.206963;
   DATA[1842,13] := 791.4637;
   DATA[1842,14] := 1.0;
   DATA[1842,15] := 2.0;
   DATA[1842,16] := 1.0;
   DATA[1842,17] := 1.0;
   DATA[1842,18] := 1.0;
   DATA[1842,19] := 2.0;
   DATA[1842,20] := 148.808;
   DATA[1842,21] := 154.3707;
   DATA[1842,22] := 1.714798;
   DATA[1842,23] := 815.4063;
   DATA[1842,24] := 2.0;
   DATA[1842,25] := 2.0;
   DATA[1842,26] := 7.874135;
   DATA[1842,27] := 143.4504;
   DATA[1842,28] := 262.3686;
   DATA[1842,29] := 11.92002;
   DATA[1842,30] := 1.722123;
   DATA[1842,31] := 1.30178;
   DATA[1842,32] := 0.7355248;
   DATA[1842,33] := 0.3084905;
   DATA[1842,34] := 2.0;
   DATA[1842,35] := 249.9519;
   DATA[1842,36] := 1.69801;
   DATA[1842,37] := 188.7657;
   DATA[1842,38] := 0.000128152;
   DATA[1842,39] := 1.0;
   DATA[1842,40] := 1.0;
   DATA[1843,0] := 2.590398;
   DATA[1843,1] := 858.8503;
   DATA[1843,2] := 2.0;
   DATA[1843,3] := 2.0;
   DATA[1843,4] := 265.0282;
   DATA[1843,5] := 8.449949;
   DATA[1843,6] := 325.455;
   DATA[1843,7] := 2.418736;
   DATA[1843,8] := 2.0;
   DATA[1843,9] := 2.0;
   DATA[1843,10] := 2.0;
   DATA[1843,11] := 19.69076;
   DATA[1843,12] := 2.205426;
   DATA[1843,13] := 790.7828;
   DATA[1843,14] := 1.0;
   DATA[1843,15] := 2.0;
   DATA[1843,16] := 1.0;
   DATA[1843,17] := 1.0;
   DATA[1843,18] := 1.0;
   DATA[1843,19] := 2.0;
   DATA[1843,20] := 148.808;
   DATA[1843,21] := 154.3707;
   DATA[1843,22] := 1.714798;
   DATA[1843,23] := 815.4448;
   DATA[1843,24] := 2.0;
   DATA[1843,25] := 2.0;
   DATA[1843,26] := 7.874135;
   DATA[1843,27] := 143.5529;
   DATA[1843,28] := 262.3686;
   DATA[1843,29] := 11.92002;
   DATA[1843,30] := 1.723148;
   DATA[1843,31] := 1.294479;
   DATA[1843,32] := 0.7355248;
   DATA[1843,33] := 0.3084905;
   DATA[1843,34] := 2.0;
   DATA[1843,35] := 249.9519;
   DATA[1843,36] := 1.69801;
   DATA[1843,37] := 188.9419;
   DATA[1843,38] := 0.000128152;
   DATA[1843,39] := 1.0;
   DATA[1843,40] := 1.0;
   DATA[1844,0] := 2.572142;
   DATA[1844,1] := 858.8896;
   DATA[1844,2] := 2.0;
   DATA[1844,3] := 2.0;
   DATA[1844,4] := 265.1884;
   DATA[1844,5] := 8.443541;
   DATA[1844,6] := 326.5829;
   DATA[1844,7] := 2.441034;
   DATA[1844,8] := 2.0;
   DATA[1844,9] := 2.0;
   DATA[1844,10] := 2.0;
   DATA[1844,11] := 19.69076;
   DATA[1844,12] := 2.207091;
   DATA[1844,13] := 790.5024;
   DATA[1844,14] := 1.0;
   DATA[1844,15] := 2.0;
   DATA[1844,16] := 1.0;
   DATA[1844,17] := 1.0;
   DATA[1844,18] := 1.0;
   DATA[1844,19] := 2.0;
   DATA[1844,20] := 148.808;
   DATA[1844,21] := 154.3707;
   DATA[1844,22] := 1.714798;
   DATA[1844,23] := 815.5217;
   DATA[1844,24] := 2.0;
   DATA[1844,25] := 2.0;
   DATA[1844,26] := 7.874135;
   DATA[1844,27] := 143.5529;
   DATA[1844,28] := 262.3686;
   DATA[1844,29] := 11.92002;
   DATA[1844,30] := 1.724045;
   DATA[1844,31] := 1.274497;
   DATA[1844,32] := 0.7355248;
   DATA[1844,33] := 0.3084905;
   DATA[1844,34] := 2.0;
   DATA[1844,35] := 249.9519;
   DATA[1844,36] := 1.69801;
   DATA[1844,37] := 188.9419;
   DATA[1844,38] := 0.000128152;
   DATA[1844,39] := 1.0;
   DATA[1844,40] := 1.0;
   DATA[1845,0] := 2.559651;
   DATA[1845,1] := 859.1644;
   DATA[1845,2] := 2.0;
   DATA[1845,3] := 2.0;
   DATA[1845,4] := 265.1884;
   DATA[1845,5] := 8.439375;
   DATA[1845,6] := 327.7365;
   DATA[1845,7] := 2.462179;
   DATA[1845,8] := 2.0;
   DATA[1845,9] := 2.0;
   DATA[1845,10] := 2.0;
   DATA[1845,11] := 19.65555;
   DATA[1845,12] := 2.208372;
   DATA[1845,13] := 790.2621;
   DATA[1845,14] := 1.0;
   DATA[1845,15] := 2.0;
   DATA[1845,16] := 1.0;
   DATA[1845,17] := 1.0;
   DATA[1845,18] := 1.0;
   DATA[1845,19] := 2.0;
   DATA[1845,20] := 148.808;
   DATA[1845,21] := 154.3707;
   DATA[1845,22] := 1.714798;
   DATA[1845,23] := 815.1371;
   DATA[1845,24] := 2.0;
   DATA[1845,25] := 2.0;
   DATA[1845,26] := 7.874135;
   DATA[1845,27] := 143.5529;
   DATA[1845,28] := 262.3686;
   DATA[1845,29] := 12.26609;
   DATA[1845,30] := 1.724301;
   DATA[1845,31] := 1.271295;
   DATA[1845,32] := 0.7355248;
   DATA[1845,33] := 0.3074656;
   DATA[1845,34] := 2.0;
   DATA[1845,35] := 249.9519;
   DATA[1845,36] := 1.69801;
   DATA[1845,37] := 188.9419;
   DATA[1845,38] := 0.000128152;
   DATA[1845,39] := 1.0;
   DATA[1845,40] := 1.0;
   DATA[1846,0] := 2.542356;
   DATA[1846,1] := 859.5176;
   DATA[1846,2] := 2.0;
   DATA[1846,3] := 2.0;
   DATA[1846,4] := 264.2592;
   DATA[1846,5] := 8.434889;
   DATA[1846,6] := 328.7618;
   DATA[1846,7] := 2.46487;
   DATA[1846,8] := 2.0;
   DATA[1846,9] := 2.0;
   DATA[1846,10] := 2.0;
   DATA[1846,11] := 19.68436;
   DATA[1846,12] := 2.208372;
   DATA[1846,13] := 790.182;
   DATA[1846,14] := 1.0;
   DATA[1846,15] := 2.0;
   DATA[1846,16] := 1.0;
   DATA[1846,17] := 1.0;
   DATA[1846,18] := 1.0;
   DATA[1846,19] := 2.0;
   DATA[1846,20] := 148.808;
   DATA[1846,21] := 154.3707;
   DATA[1846,22] := 1.715439;
   DATA[1846,23] := 815.4063;
   DATA[1846,24] := 2.0;
   DATA[1846,25] := 2.0;
   DATA[1846,26] := 7.874135;
   DATA[1846,27] := 143.5529;
   DATA[1846,28] := 262.3686;
   DATA[1846,29] := 12.26609;
   DATA[1846,30] := 1.724686;
   DATA[1846,31] := 1.271295;
   DATA[1846,32] := 0.7355248;
   DATA[1846,33] := 0.3063127;
   DATA[1846,34] := 2.0;
   DATA[1846,35] := 250.0961;
   DATA[1846,36] := 1.69801;
   DATA[1846,37] := 188.9419;
   DATA[1846,38] := 0.000128152;
   DATA[1846,39] := 1.0;
   DATA[1846,40] := 1.0;
   DATA[1847,0] := 2.525702;
   DATA[1847,1] := 859.6354;
   DATA[1847,2] := 2.0;
   DATA[1847,3] := 2.0;
   DATA[1847,4] := 263.8105;
   DATA[1847,5] := 8.429762;
   DATA[1847,6] := 329.6591;
   DATA[1847,7] := 2.466665;
   DATA[1847,8] := 2.0;
   DATA[1847,9] := 2.0;
   DATA[1847,10] := 2.0;
   DATA[1847,11] := 19.72277;
   DATA[1847,12] := 2.209397;
   DATA[1847,13] := 790.2621;
   DATA[1847,14] := 1.0;
   DATA[1847,15] := 2.0;
   DATA[1847,16] := 1.0;
   DATA[1847,17] := 1.0;
   DATA[1847,18] := 1.0;
   DATA[1847,19] := 2.0;
   DATA[1847,20] := 148.808;
   DATA[1847,21] := 154.3707;
   DATA[1847,22] := 1.715567;
   DATA[1847,23] := 815.5601;
   DATA[1847,24] := 2.0;
   DATA[1847,25] := 2.0;
   DATA[1847,26] := 7.874135;
   DATA[1847,27] := 143.5529;
   DATA[1847,28] := 262.3686;
   DATA[1847,29] := 12.26609;
   DATA[1847,30] := 1.725455;
   DATA[1847,31] := 1.271295;
   DATA[1847,32] := 0.7355248;
   DATA[1847,33] := 0.3063127;
   DATA[1847,34] := 2.0;
   DATA[1847,35] := 250.0961;
   DATA[1847,36] := 1.69801;
   DATA[1847,37] := 188.9419;
   DATA[1847,38] := 0.000128152;
   DATA[1847,39] := 1.0;
   DATA[1847,40] := 1.0;
   DATA[1848,0] := 2.510329;
   DATA[1848,1] := 860.1457;
   DATA[1848,2] := 2.0;
   DATA[1848,3] := 2.0;
   DATA[1848,4] := 263.8105;
   DATA[1848,5] := 8.425276;
   DATA[1848,6] := 330.5306;
   DATA[1848,7] := 2.466665;
   DATA[1848,8] := 2.0;
   DATA[1848,9] := 2.0;
   DATA[1848,10] := 2.0;
   DATA[1848,11] := 19.73238;
   DATA[1848,12] := 2.209397;
   DATA[1848,13] := 790.3823;
   DATA[1848,14] := 1.0;
   DATA[1848,15] := 2.0;
   DATA[1848,16] := 1.0;
   DATA[1848,17] := 1.0;
   DATA[1848,18] := 1.0;
   DATA[1848,19] := 2.0;
   DATA[1848,20] := 148.808;
   DATA[1848,21] := 154.3707;
   DATA[1848,22] := 1.716721;
   DATA[1848,23] := 815.5986;
   DATA[1848,24] := 2.0;
   DATA[1848,25] := 2.0;
   DATA[1848,26] := 7.874135;
   DATA[1848,27] := 143.5529;
   DATA[1848,28] := 262.3686;
   DATA[1848,29] := 12.26609;
   DATA[1848,30] := 1.725455;
   DATA[1848,31] := 1.280646;
   DATA[1848,32] := 0.7355248;
   DATA[1848,33] := 0.3079781;
   DATA[1848,34] := 2.0;
   DATA[1848,35] := 250.0961;
   DATA[1848,36] := 1.69801;
   DATA[1848,37] := 188.9419;
   DATA[1848,38] := 0.000128152;
   DATA[1848,39] := 1.0;
   DATA[1848,40] := 1.0;
   DATA[1849,0] := 2.499439;
   DATA[1849,1] := 859.7139;
   DATA[1849,2] := 2.0;
   DATA[1849,3] := 2.0;
   DATA[1849,4] := 263.8105;
   DATA[1849,5] := 8.42111;
   DATA[1849,6] := 330.9921;
   DATA[1849,7] := 2.466665;
   DATA[1849,8] := 2.0;
   DATA[1849,9] := 2.0;
   DATA[1849,10] := 2.0;
   DATA[1849,11] := 19.76759;
   DATA[1849,12] := 2.209397;
   DATA[1849,13] := 790.1019;
   DATA[1849,14] := 1.0;
   DATA[1849,15] := 2.0;
   DATA[1849,16] := 1.0;
   DATA[1849,17] := 1.0;
   DATA[1849,18] := 1.0;
   DATA[1849,19] := 2.0;
   DATA[1849,20] := 148.808;
   DATA[1849,21] := 154.3707;
   DATA[1849,22] := 1.717489;
   DATA[1849,23] := 815.5601;
   DATA[1849,24] := 2.0;
   DATA[1849,25] := 2.0;
   DATA[1849,26] := 7.874135;
   DATA[1849,27] := 143.5529;
   DATA[1849,28] := 262.3686;
   DATA[1849,29] := 12.26609;
   DATA[1849,30] := 1.725455;
   DATA[1849,31] := 1.276675;
   DATA[1849,32] := 0.7355248;
   DATA[1849,33] := 0.3086827;
   DATA[1849,34] := 2.0;
   DATA[1849,35] := 250.0961;
   DATA[1849,36] := 1.69801;
   DATA[1849,37] := 188.9419;
   DATA[1849,38] := 0.000128152;
   DATA[1849,39] := 1.0;
   DATA[1849,40] := 1.0;
   DATA[1850,0] := 2.481504;
   DATA[1850,1] := 859.8709;
   DATA[1850,2] := 2.0;
   DATA[1850,3] := 2.0;
   DATA[1850,4] := 264.3232;
   DATA[1850,5] := 8.416304;
   DATA[1850,6] := 331.5047;
   DATA[1850,7] := 2.466665;
   DATA[1850,8] := 2.0;
   DATA[1850,9] := 2.0;
   DATA[1850,10] := 2.0;
   DATA[1850,11] := 19.76759;
   DATA[1850,12] := 2.209397;
   DATA[1850,13] := 789.9417;
   DATA[1850,14] := 1.0;
   DATA[1850,15] := 2.0;
   DATA[1850,16] := 1.0;
   DATA[1850,17] := 1.0;
   DATA[1850,18] := 1.0;
   DATA[1850,19] := 2.0;
   DATA[1850,20] := 148.808;
   DATA[1850,21] := 154.3707;
   DATA[1850,22] := 1.717489;
   DATA[1850,23] := 816.1369;
   DATA[1850,24] := 2.0;
   DATA[1850,25] := 2.0;
   DATA[1850,26] := 7.874135;
   DATA[1850,27] := 143.5529;
   DATA[1850,28] := 262.3686;
   DATA[1850,29] := 12.22763;
   DATA[1850,30] := 1.725455;
   DATA[1850,31] := 1.271039;
   DATA[1850,32] := 0.7355248;
   DATA[1850,33] := 0.3086827;
   DATA[1850,34] := 2.0;
   DATA[1850,35] := 250.0961;
   DATA[1850,36] := 1.69801;
   DATA[1850,37] := 188.9419;
   DATA[1850,38] := 0.000128152;
   DATA[1850,39] := 1.0;
   DATA[1850,40] := 1.0;
   DATA[1851,0] := 2.469654;
   DATA[1851,1] := 860.1064;
   DATA[1851,2] := 2.0;
   DATA[1851,3] := 2.0;
   DATA[1851,4] := 264.3232;
   DATA[1851,5] := 8.414381;
   DATA[1851,6] := 331.8893;
   DATA[1851,7] := 2.466665;
   DATA[1851,8] := 2.0;
   DATA[1851,9] := 2.0;
   DATA[1851,10] := 2.0;
   DATA[1851,11] := 19.73878;
   DATA[1851,12] := 2.207091;
   DATA[1851,13] := 790.5024;
   DATA[1851,14] := 1.0;
   DATA[1851,15] := 2.0;
   DATA[1851,16] := 1.0;
   DATA[1851,17] := 1.0;
   DATA[1851,18] := 1.0;
   DATA[1851,19] := 2.0;
   DATA[1851,20] := 148.808;
   DATA[1851,21] := 154.3707;
   DATA[1851,22] := 1.717489;
   DATA[1851,23] := 816.483;
   DATA[1851,24] := 2.0;
   DATA[1851,25] := 2.0;
   DATA[1851,26] := 7.874135;
   DATA[1851,27] := 143.5529;
   DATA[1851,28] := 262.3686;
   DATA[1851,29] := 12.22763;
   DATA[1851,30] := 1.725455;
   DATA[1851,31] := 1.276803;
   DATA[1851,32] := 0.7355248;
   DATA[1851,33] := 0.3086186;
   DATA[1851,34] := 2.0;
   DATA[1851,35] := 250.0961;
   DATA[1851,36] := 1.69801;
   DATA[1851,37] := 188.9419;
   DATA[1851,38] := 0.000128152;
   DATA[1851,39] := 1.0;
   DATA[1851,40] := 1.0;
   DATA[1852,0] := 2.450758;
   DATA[1852,1] := 860.4597;
   DATA[1852,2] := 2.0;
   DATA[1852,3] := 2.0;
   DATA[1852,4] := 264.3232;
   DATA[1852,5] := 8.410856;
   DATA[1852,6] := 332.3507;
   DATA[1852,7] := 2.466665;
   DATA[1852,8] := 2.0;
   DATA[1852,9] := 2.0;
   DATA[1852,10] := 2.0;
   DATA[1852,11] := 19.72277;
   DATA[1852,12] := 2.207091;
   DATA[1852,13] := 790.2621;
   DATA[1852,14] := 1.0;
   DATA[1852,15] := 2.0;
   DATA[1852,16] := 1.0;
   DATA[1852,17] := 1.0;
   DATA[1852,18] := 1.0;
   DATA[1852,19] := 2.0;
   DATA[1852,20] := 148.808;
   DATA[1852,21] := 154.4476;
   DATA[1852,22] := 1.717489;
   DATA[1852,23] := 817.1367;
   DATA[1852,24] := 2.0;
   DATA[1852,25] := 2.0;
   DATA[1852,26] := 7.874135;
   DATA[1852,27] := 143.5529;
   DATA[1852,28] := 262.3686;
   DATA[1852,29] := 12.22763;
   DATA[1852,30] := 1.724173;
   DATA[1852,31] := 1.281927;
   DATA[1852,32] := 0.7355248;
   DATA[1852,33] := 0.3084265;
   DATA[1852,34] := 2.0;
   DATA[1852,35] := 250.0961;
   DATA[1852,36] := 1.69801;
   DATA[1852,37] := 188.9419;
   DATA[1852,38] := 0.000128152;
   DATA[1852,39] := 1.0;
   DATA[1852,40] := 1.0;
   DATA[1853,0] := 2.437946;
   DATA[1853,1] := 860.499;
   DATA[1853,2] := 2.0;
   DATA[1853,3] := 2.0;
   DATA[1853,4] := 263.8426;
   DATA[1853,5] := 8.407652;
   DATA[1853,6] := 332.6327;
   DATA[1853,7] := 2.465767;
   DATA[1853,8] := 2.0;
   DATA[1853,9] := 2.0;
   DATA[1853,10] := 2.0;
   DATA[1853,11] := 19.69076;
   DATA[1853,12] := 2.207091;
   DATA[1853,13] := 790.142;
   DATA[1853,14] := 1.0;
   DATA[1853,15] := 2.0;
   DATA[1853,16] := 1.0;
   DATA[1853,17] := 1.0;
   DATA[1853,18] := 1.0;
   DATA[1853,19] := 2.0;
   DATA[1853,20] := 148.808;
   DATA[1853,21] := 154.4476;
   DATA[1853,22] := 1.717489;
   DATA[1853,23] := 817.4443;
   DATA[1853,24] := 2.0;
   DATA[1853,25] := 2.0;
   DATA[1853,26] := 7.874135;
   DATA[1853,27] := 143.5529;
   DATA[1853,28] := 262.3686;
   DATA[1853,29] := 12.22763;
   DATA[1853,30] := 1.723789;
   DATA[1853,31] := 1.281927;
   DATA[1853,32] := 0.7355248;
   DATA[1853,33] := 0.3084265;
   DATA[1853,34] := 2.0;
   DATA[1853,35] := 250.0961;
   DATA[1853,36] := 1.69801;
   DATA[1853,37] := 188.9419;
   DATA[1853,38] := 0.000128152;
   DATA[1853,39] := 1.0;
   DATA[1853,40] := 1.0;
   DATA[1854,0] := 2.427377;
   DATA[1854,1] := 860.6559;
   DATA[1854,2] := 2.0;
   DATA[1854,3] := 2.0;
   DATA[1854,4] := 263.8426;
   DATA[1854,5] := 8.403486;
   DATA[1854,6] := 332.889;
   DATA[1854,7] := 2.46423;
   DATA[1854,8] := 2.0;
   DATA[1854,9] := 2.0;
   DATA[1854,10] := 2.0;
   DATA[1854,11] := 19.69076;
   DATA[1854,12] := 2.207091;
   DATA[1854,13] := 789.7014;
   DATA[1854,14] := 1.0;
   DATA[1854,15] := 2.0;
   DATA[1854,16] := 1.0;
   DATA[1854,17] := 1.0;
   DATA[1854,18] := 1.0;
   DATA[1854,19] := 2.0;
   DATA[1854,20] := 148.808;
   DATA[1854,21] := 154.4476;
   DATA[1854,22] := 1.716592;
   DATA[1854,23] := 817.4827;
   DATA[1854,24] := 2.0;
   DATA[1854,25] := 2.0;
   DATA[1854,26] := 7.874135;
   DATA[1854,27] := 143.5529;
   DATA[1854,28] := 262.3686;
   DATA[1854,29] := 12.15073;
   DATA[1854,30] := 1.722763;
   DATA[1854,31] := 1.281927;
   DATA[1854,32] := 0.7355248;
   DATA[1854,33] := 0.3084265;
   DATA[1854,34] := 2.0;
   DATA[1854,35] := 250.0961;
   DATA[1854,36] := 1.69801;
   DATA[1854,37] := 188.9419;
   DATA[1854,38] := 0.000128152;
   DATA[1854,39] := 1.0;
   DATA[1854,40] := 1.0;
   DATA[1855,0] := 2.426416;
   DATA[1855,1] := 860.5382;
   DATA[1855,2] := 2.0;
   DATA[1855,3] := 2.0;
   DATA[1855,4] := 263.6824;
   DATA[1855,5] := 8.403486;
   DATA[1855,6] := 332.9915;
   DATA[1855,7] := 2.46423;
   DATA[1855,8] := 2.0;
   DATA[1855,9] := 2.0;
   DATA[1855,10] := 2.0;
   DATA[1855,11] := 19.75799;
   DATA[1855,12] := 2.207091;
   DATA[1855,13] := 789.9017;
   DATA[1855,14] := 1.0;
   DATA[1855,15] := 2.0;
   DATA[1855,16] := 1.0;
   DATA[1855,17] := 1.0;
   DATA[1855,18] := 1.0;
   DATA[1855,19] := 2.0;
   DATA[1855,20] := 148.808;
   DATA[1855,21] := 154.4476;
   DATA[1855,22] := 1.713261;
   DATA[1855,23] := 817.6749;
   DATA[1855,24] := 2.0;
   DATA[1855,25] := 2.0;
   DATA[1855,26] := 7.874135;
   DATA[1855,27] := 143.5529;
   DATA[1855,28] := 262.3686;
   DATA[1855,29] := 12.15073;
   DATA[1855,30] := 1.722763;
   DATA[1855,31] := 1.281927;
   DATA[1855,32] := 0.7355248;
   DATA[1855,33] := 0.3084265;
   DATA[1855,34] := 2.0;
   DATA[1855,35] := 250.0961;
   DATA[1855,36] := 1.69801;
   DATA[1855,37] := 188.9419;
   DATA[1855,38] := 0.000128152;
   DATA[1855,39] := 1.0;
   DATA[1855,40] := 1.0;
   DATA[1856,0] := 2.434744;
   DATA[1856,1] := 860.3027;
   DATA[1856,2] := 2.0;
   DATA[1856,3] := 2.0;
   DATA[1856,4] := 263.362;
   DATA[1856,5] := 8.399641;
   DATA[1856,6] := 333.1197;
   DATA[1856,7] := 2.466665;
   DATA[1856,8] := 2.0;
   DATA[1856,9] := 2.0;
   DATA[1856,10] := 2.0;
   DATA[1856,11] := 19.76439;
   DATA[1856,12] := 2.207091;
   DATA[1856,13] := 790.2621;
   DATA[1856,14] := 1.0;
   DATA[1856,15] := 2.0;
   DATA[1856,16] := 1.0;
   DATA[1856,17] := 1.0;
   DATA[1856,18] := 1.0;
   DATA[1856,19] := 2.0;
   DATA[1856,20] := 148.808;
   DATA[1856,21] := 154.4476;
   DATA[1856,22] := 1.713261;
   DATA[1856,23] := 817.9056;
   DATA[1856,24] := 2.0;
   DATA[1856,25] := 2.0;
   DATA[1856,26] := 7.874135;
   DATA[1856,27] := 143.5529;
   DATA[1856,28] := 262.3686;
   DATA[1856,29] := 12.15073;
   DATA[1856,30] := 1.721738;
   DATA[1856,31] := 1.275138;
   DATA[1856,32] := 0.7355248;
   DATA[1856,33] := 0.3084265;
   DATA[1856,34] := 2.0;
   DATA[1856,35] := 250.0961;
   DATA[1856,36] := 1.69801;
   DATA[1856,37] := 188.8939;
   DATA[1856,38] := 0.000128152;
   DATA[1856,39] := 1.0;
   DATA[1856,40] := 1.0;
   DATA[1857,0] := 2.487589;
   DATA[1857,1] := 860.9307;
   DATA[1857,2] := 2.0;
   DATA[1857,3] := 2.0;
   DATA[1857,4] := 263.362;
   DATA[1857,5] := 8.398359;
   DATA[1857,6] := 333.171;
   DATA[1857,7] := 2.469228;
   DATA[1857,8] := 2.0;
   DATA[1857,9] := 2.0;
   DATA[1857,10] := 2.0;
   DATA[1857,11] := 19.76759;
   DATA[1857,12] := 2.208756;
   DATA[1857,13] := 790.182;
   DATA[1857,14] := 1.0;
   DATA[1857,15] := 2.0;
   DATA[1857,16] := 1.0;
   DATA[1857,17] := 1.0;
   DATA[1857,18] := 1.0;
   DATA[1857,19] := 2.0;
   DATA[1857,20] := 148.808;
   DATA[1857,21] := 154.4476;
   DATA[1857,22] := 1.711723;
   DATA[1857,23] := 817.9441;
   DATA[1857,24] := 2.0;
   DATA[1857,25] := 2.0;
   DATA[1857,26] := 7.874135;
   DATA[1857,27] := 143.5529;
   DATA[1857,28] := 262.3686;
   DATA[1857,29] := 12.15073;
